KUKA KRL program: MyProgram_106().src

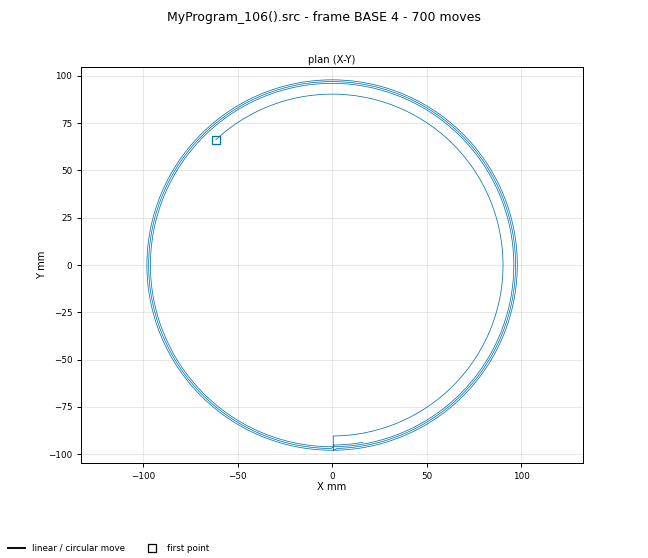
[picture p0: tool path of MyProgram_106().src in frame BASE 4, 700 of 700 moves have a stored position in this frame; points joined in program order, loops and branches not executed]
&ACCESS RVP
&REL 1
&PARAM TEMPLATE = C:\KRC\Roboter\Template\vorgabe
&PARAM EDITMASK = *
DEF MyProgram_106()
; ---- Setting reference (Base) ----
$BASE = BASE_DATA[4]

; --------------------------
; ---- Setting tool (TCP) ----
$TOOL = TOOL_DATA[3]
; --------------------------

$VEL.CP = VEL_APROX_PRINT
Startdeposition()
$VEL.CP = VEL_PRINT
LIN {X -61.5081,Y 66.2185,Z 94,A 127.1384,B 24.9108,C -2.1806,E1 24.8923,E2 -42.0687} C_DIS
LIN {X -59.0339,Y 68.4334,Z 94,A 125.0218,B 24.9104,C -2.1851,E1 24.8968,E2 -39.9543} C_DIS
LIN {X -56.4801,Y 70.5559,Z 94,A 122.9034,B 24.9101,C -2.1892,E1 24.9013,E2 -37.8379} C_DIS
LIN {X -54.0546,Y 72.4294,Z 94,A 121.1393,B 24.9093,C -2.1987,E1 24.9052,E2 -36.09} C_DIS
LIN {X -51.3564,Y 74.3668,Z 94,A 119.0568,B 24.9089,C -2.2037,E1 24.91,E2 -34.012} C_DIS
LIN {X -49.519,Y 75.6028,Z 94,A 117.6469,B 24.9087,C -2.2062,E1 24.9132,E2 -32.6035} C_DIS
LIN {X -47.5461,Y 76.8594,Z 94,A 115.9946,B 24.9089,C -2.2038,E1 24.9172,E2 -30.9403} C_DIS
LIN {X -44.7585,Y 78.515,Z 94,A 113.9269,B 24.9086,C -2.2071,E1 24.9222,E2 -28.8743} C_DIS
LIN {X -41.8485,Y 80.1038,Z 94,A 111.9477,B 24.908,C -2.2144,E1 24.927,E2 -26.9069} C_DIS
LIN {X -39.6316,Y 81.2248,Z 94,A 110.4097,B 24.9077,C -2.218,E1 24.9308,E2 -25.3735} C_DIS
LIN {X -36.8751,Y 82.5114,Z 94,A 108.4363,B 24.9076,C -2.2196,E1 24.9358,E2 -23.3989} C_DIS
LIN {X -34.5929,Y 83.4953,Z 94,A 106.888,B 24.9073,C -2.2227,E1 24.9398,E2 -21.8544} C_DIS
LIN {X -32.7956,Y 84.2161,Z 94,A 105.623,B 24.9073,C -2.2232,E1 24.9431,E2 -20.5879} C_DIS
LIN {X -29.6593,Y 85.3712,Z 94,A 103.3582,B 24.9074,C -2.2214,E1 24.9491,E2 -18.3142} C_DIS
LIN {X -26.4788,Y 86.4106,Z 94,A 101.4259,B 24.9067,C -2.2297,E1 24.9542,E2 -16.3983} C_DIS
LIN {X -24.0911,Y 87.1077,Z 94,A 99.8258,B 24.9067,C -2.2306,E1 24.9585,E2 -14.7978} C_DIS
LIN {X -21.1443,Y 87.8683,Z 94,A 97.8908,B 24.9065,C -2.2324,E1 24.9637,E2 -12.8641} C_DIS
LIN {X -18.7193,Y 88.4179,Z 94,A 96.311,B 24.9065,C -2.2336,E1 24.968,E2 -11.2853} C_DIS
LIN {X -16.8191,Y 88.7977,Z 94,A 95.0427,B 24.9065,C -2.2334,E1 24.9715,E2 -10.015} C_DIS
LIN {X -14.6242,Y 89.1855,Z 94,A 93.4958,B 24.9067,C -2.2302,E1 24.9758,E2 -8.4591} C_DIS
LIN {X -11.3226,Y 89.6645,Z 94,A 91.5124,B 24.9062,C -2.2356,E1 24.9812,E2 -6.4871} C_DIS
LIN {X -8.8533,Y 89.9431,Z 94,A 89.9727,B 24.9061,C -2.2376,E1 24.9855,E2 -4.9513} C_DIS
LIN {X -6.6558,Y 90.1323,Z 94,A 88.571,B 24.9061,C -2.2381,E1 24.9894,E2 -3.5501} C_DIS
LIN {X -4.1214,Y 90.2824,Z 94,A 86.8039,B 24.9064,C -2.2337,E1 24.9944,E2 -1.772} C_DIS
LIN {X -1.0898,Y 90.3711,Z 94,A 84.8009,B 24.9066,C -2.2316,E1 25,E2 0.2361} C_DIS
LIN {X 2.2165,Y 90.3505,Z 94,A 82.9393,B 24.9059,C -2.2394,E1 25.0051,E2 2.0789} C_DIS
LIN {X 5.279,Y 90.2222,Z 94,A 80.9608,B 24.906,C -2.2384,E1 25.0106,E2 4.0591} C_DIS
LIN {X 8.157,Y 90.0073,Z 94,A 79.047,B 24.9062,C -2.2356,E1 25.016,E2 5.9787} C_DIS
LIN {X 10.7987,Y 89.7291,Z 94,A 77.4482,B 24.906,C -2.2381,E1 25.0204,E2 7.5704} C_DIS
LIN {X 12.992,Y 89.4378,Z 94,A 75.9187,B 24.9064,C -2.2336,E1 25.0246,E2 9.1093} C_DIS
LIN {X 16.1999,Y 88.9125,Z 94,A 73.9645,B 24.9062,C -2.2363,E1 25.03,E2 11.0548} C_DIS
LIN {X 19.5413,Y 88.2386,Z 94,A 71.8741,B 24.9061,C -2.2377,E1 25.0357,E2 13.1395} C_DIS
LIN {X 21.9634,Y 87.6684,Z 94,A 70.2868,B 24.9061,C -2.2364,E1 25.04,E2 14.7274} C_DIS
LIN {X 24.9051,Y 86.8772,Z 94,A 68.3251,B 24.9064,C -2.2342,E1 25.0453,E2 16.6913} C_DIS
LIN {X 27.5626,Y 86.071,Z 94,A 66.4674,B 24.9067,C -2.2296,E1 25.0503,E2 18.5565} C_DIS
LIN {X 30.7614,Y 84.9801,Z 94,A 64.315,B 24.9069,C -2.2274,E1 25.0559,E2 20.7098} C_DIS
LIN {X 33.4831,Y 83.946,Z 94,A 62.6281,B 24.9066,C -2.2309,E1 25.0603,E2 22.3847} C_DIS
LIN {X 35.6162,Y 83.0639,Z 94,A 60.9576,B 24.9074,C -2.2224,E1 25.0646,E2 24.0714} C_DIS
LIN {X 38.6404,Y 81.701,Z 94,A 59.0613,B 24.907,C -2.2269,E1 25.0694,E2 25.9522} C_DIS
LIN {X 41.3681,Y 80.3529,Z 94,A 57.1008,B 24.9073,C -2.2234,E1 25.0743,E2 27.9156} C_DIS
LIN {X 43.3395,Y 79.307,Z 94,A 55.5648,B 24.9078,C -2.2174,E1 25.0781,E2 29.4615} C_DIS
LIN {X 46.2751,Y 77.6309,Z 94,A 53.5477,B 24.9077,C -2.2186,E1 25.083,E2 31.4697} C_DIS
LIN {X 48.3763,Y 76.3403,Z 94,A 52.0379,B 24.9077,C -2.218,E1 25.0865,E2 32.9761} C_DIS
LIN {X 50.2205,Y 75.1401,Z 94,A 50.6472,B 24.9079,C -2.2159,E1 25.0898,E2 34.367} C_DIS
LIN {X 52.2581,Y 73.7361,Z 94,A 48.9167,B 24.9086,C -2.2078,E1 25.0938,E2 36.1109} C_DIS
LIN {X 54.6991,Y 71.9452,Z 94,A 46.9487,B 24.909,C -2.2027,E1 25.0982,E2 38.0837} C_DIS
LIN {X 57.3349,Y 69.8631,Z 94,A 44.8265,B 24.9093,C -2.199,E1 25.1028,E2 40.2067} C_DIS
LIN {X 59.8757,Y 67.698,Z 94,A 42.7258,B 24.9096,C -2.1954,E1 25.1072,E2 42.3076} C_DIS
LIN {X 62.3215,Y 65.4535,Z 94,A 40.629,B 24.9099,C -2.1914,E1 25.1115,E2 44.4054} C_DIS
LIN {X 64.6833,Y 63.1206,Z 94,A 38.534,B 24.9103,C -2.1872,E1 25.1156,E2 46.5013} C_DIS
LIN {X 66.9576,Y 60.7026,Z 94,A 36.4373,B 24.9106,C -2.1828,E1 25.1196,E2 48.5992} C_DIS
LIN {X 69.1579,Y 58.1834,Z 94,A 34.3106,B 24.911,C -2.1777,E1 25.1235,E2 50.7283} C_DIS
LIN {X 71.2845,Y 55.5572,Z 94,A 32.1828,B 24.9114,C -2.1731,E1 25.1271,E2 52.8571} C_DIS
LIN {X 73.4267,Y 52.6916,Z 94,A 30.0253,B 24.9116,C -2.1714,E1 25.1307,E2 55.0081} C_DIS
LIN {X 74.9959,Y 50.4334,Z 94,A 28.4236,B 24.9116,C -2.172,E1 25.1332,E2 56.6006} C_DIS
LIN {X 76.2091,Y 48.5808,Z 94,A 27.0277,B 24.9118,C -2.1687,E1 25.1353,E2 57.9974} C_DIS
LIN {X 77.3765,Y 46.6989,Z 94,A 25.6013,B 24.9122,C -2.1642,E1 25.1374,E2 59.4271} C_DIS
LIN {X 78.5152,Y 44.7582,Z 94,A 24.0499,B 24.9128,C -2.1559,E1 25.1396,E2 60.99} C_DIS
LIN {X 80.1014,Y 41.8532,Z 94,A 22.1266,B 24.9128,C -2.1564,E1 25.1421,E2 62.902} C_DIS
LIN {X 81.2217,Y 39.638,Z 94,A 20.3536,B 24.9137,C -2.1449,E1 25.1443,E2 64.6927} C_DIS
LIN {X 82.5072,Y 36.8844,Z 94,A 18.4926,B 24.914,C -2.1418,E1 25.1465,E2 66.5508} C_DIS
LIN {X 83.7784,Y 33.8975,Z 94,A 16.5874,B 24.914,C -2.1413,E1 25.1485,E2 68.4467} C_DIS
LIN {X 84.7137,Y 31.4916,Z 94,A 14.978,B 24.9143,C -2.1375,E1 25.1501,E2 70.0562} C_DIS
LIN {X 85.8199,Y 28.3386,Z 94,A 12.8796,B 24.9148,C -2.1319,E1 25.152,E2 72.1559} C_DIS
LIN {X 86.7244,Y 25.4319,Z 94,A 10.924,B 24.9153,C -2.1252,E1 25.1536,E2 74.1162} C_DIS
LIN {X 87.3926,Y 23.0362,Z 94,A 9.2221,B 24.916,C -2.1159,E1 25.1549,E2 75.8303} C_DIS
LIN {X 88.1253,Y 20.0464,Z 94,A 7.4136,B 24.9161,C -2.1151,E1 25.156,E2 77.6303} C_DIS
LIN {X 88.6437,Y 17.6188,Z 94,A 5.8952,B 24.9163,C -2.1122,E1 25.1569,E2 79.1467} C_DIS
LIN {X 89.0428,Y 15.4757,Z 94,A 4.5192,B 24.9167,C -2.1081,E1 25.1576,E2 80.5244} C_DIS
LIN {X 89.399,Y 13.2645,Z 94,A 3.1049,B 24.917,C -2.1038,E1 25.1582,E2 81.9404} C_DIS
LIN {X 89.6657,Y 11.3128,Z 94,A 1.8305,B 24.9174,C -2.099,E1 25.1587,E2 83.2187} C_DIS
LIN {X 89.943,Y 8.8544,Z 94,A 0.2027,B 24.9179,C -2.0918,E1 25.1591,E2 84.8538} C_DIS
LIN {X 90.197,Y 5.7001,Z 94,A -1.8462,B 24.9186,C -2.0839,E1 25.1595,E2 86.9092} C_DIS
LIN {X 90.3415,Y 2.5118,Z 94,A -3.7689,B 24.9188,C -2.0811,E1 25.1597,E2 88.8271} C_DIS
LIN {X 90.3738,Y -0.7138,Z 94,A -5.9406,B 24.9196,C -2.07,E1 25.1597,E2 91.0121} C_DIS
LIN {X 90.2796,Y -4.186,Z 94,A -7.911,B 24.9196,C -2.0712,E1 25.1596,E2 92.9678} C_DIS
LIN {X 90.1322,Y -6.657,Z 94,A -9.4653,B 24.9199,C -2.0667,E1 25.1593,E2 94.5235} C_DIS
LIN {X 89.9431,Y -8.8525,Z 94,A -10.8563,B 24.9202,C -2.0624,E1 25.1589,E2 95.9164} C_DIS
LIN {X 89.5538,Y -12.1755,Z 94,A -12.9566,B 24.9207,C -2.0564,E1 25.1582,E2 98.0186} C_DIS
LIN {X 89.0487,Y -15.4423,Z 94,A -15.0435,B 24.9212,C -2.05,E1 25.1573,E2 100.1083} C_DIS
LIN {X 88.6386,Y -17.6444,Z 94,A -16.6575,B 24.9221,C -2.0385,E1 25.1564,E2 101.7401} C_DIS
LIN {X 87.933,Y -20.8787,Z 94,A -18.6638,B 24.9223,C -2.0351,E1 25.1552,E2 103.7426} C_DIS
LIN {X 87.1809,Y -23.82,Z 94,A -20.455,B 24.9224,C -2.0339,E1 25.1539,E2 105.5265} C_DIS
LIN {X 86.4846,Y -26.2404,Z 94,A -22.0353,B 24.9228,C -2.0294,E1 25.1527,E2 107.1083} C_DIS
LIN {X 85.8159,Y -28.3509,Z 94,A -23.4299,B 24.9231,C -2.0254,E1 25.1515,E2 108.5045} C_DIS
LIN {X 85.0617,Y -30.5377,Z 94,A -24.8793,B 24.9234,C -2.0214,E1 25.1501,E2 109.955} C_DIS
LIN {X 84.199,Y -32.8392,Z 94,A -26.5824,B 24.9241,C -2.0114,E1 25.1484,E2 111.6723} C_DIS
LIN {X 83.1636,Y -35.3801,Z 94,A -28.1431,B 24.9241,C -2.0126,E1 25.1467,E2 113.2217} C_DIS
LIN {X 82.1671,Y -37.6391,Z 94,A -29.8413,B 24.9248,C -2.003,E1 25.1448,E2 114.9332} C_DIS
LIN {X 80.8611,Y -40.3655,Z 94,A -31.6269,B 24.9248,C -2.002,E1 25.1426,E2 116.7115} C_DIS
LIN {X 79.7039,Y -42.6077,Z 94,A -33.2085,B 24.9252,C -1.998,E1 25.1406,E2 118.2944} C_DIS
LIN {X 78.6361,Y -44.5478,Z 94,A -34.6056,B 24.9254,C -1.9941,E1 25.1387,E2 119.6933} C_DIS
LIN {X 77.6608,Y -46.2246,Z 94,A -35.871,B 24.9258,C -1.9893,E1 25.1369,E2 120.9635} C_DIS
LIN {X 76.3474,Y -48.3653,Z 94,A -37.6069,B 24.9265,C -1.9796,E1 25.1343,E2 122.7135} C_DIS
LIN {X 74.5206,Y -51.1353,Z 94,A -39.4997,B 24.9264,C -1.9813,E1 25.1313,E2 124.593} C_DIS
LIN {X 73.2465,Y -52.9442,Z 94,A -40.8949,B 24.9267,C -1.9777,E1 25.1291,E2 125.9899} C_DIS
LIN {X 71.5903,Y -55.1603,Z 94,A -42.7617,B 24.9273,C -1.969,E1 25.1259,E2 127.8684} C_DIS
LIN {X 69.4989,Y -57.7731,Z 94,A -44.8582,B 24.9277,C -1.9643,E1 25.1222,E2 129.9663} C_DIS
LIN {X 67.3324,Y -60.2842,Z 94,A -46.927,B 24.928,C -1.9601,E1 25.1184,E2 132.0357} C_DIS
LIN {X 65.0939,Y -62.6947,Z 94,A -49.0471,B 24.9284,C -1.9537,E1 25.1143,E2 134.1617} C_DIS
LIN {X 62.7061,Y -65.0829,Z 94,A -51.1535,B 24.9287,C -1.9497,E1 25.1101,E2 136.2685} C_DIS
LIN {X 60.2762,Y -67.3396,Z 94,A -53.2426,B 24.9291,C -1.9453,E1 25.1058,E2 138.3597} C_DIS
LIN {X 57.7644,Y -69.5061,Z 94,A -55.3481,B 24.9294,C -1.9405,E1 25.1013,E2 140.4684} C_DIS
LIN {X 55.1537,Y -71.5954,Z 94,A -57.4017,B 24.9296,C -1.9382,E1 25.0968,E2 142.5197} C_DIS
LIN {X 52.9367,Y -73.2519,Z 94,A -59.0802,B 24.9296,C -1.9372,E1 25.0931,E2 144.1946} C_DIS
LIN {X 50.4391,Y -74.9921,Z 94,A -61.0056,B 24.9299,C -1.9335,E1 25.0886,E2 146.1223} C_DIS
LIN {X 48.5883,Y -76.2043,Z 94,A -62.4025,B 24.9301,C -1.931,E1 25.0854,E2 147.5205} C_DIS
LIN {X 46.7085,Y -77.3707,Z 94,A -63.8378,B 24.9304,C -1.9272,E1 25.0819,E2 148.9603} C_DIS
LIN {X 44.7808,Y -78.5022,Z 94,A -65.3722,B 24.9308,C -1.9206,E1 25.0782,E2 150.5057} C_DIS
LIN {X 41.7682,Y -80.1461,Z 94,A -67.5477,B 24.9311,C -1.9168,E1 25.0728,E2 152.6839} C_DIS
LIN {X 38.8458,Y -81.6023,Z 94,A -69.4397,B 24.9309,C -1.9197,E1 25.0681,E2 154.5642} C_DIS
LIN {X 36.8543,Y -82.5208,Z 94,A -70.8602,B 24.9311,C -1.9165,E1 25.0645,E2 155.9887} C_DIS
LIN {X 34.7762,Y -83.418,Z 94,A -72.2755,B 24.9312,C -1.915,E1 25.0609,E2 157.404} C_DIS
LIN {X 32.799,Y -84.2148,Z 94,A -73.6475,B 24.9314,C -1.9125,E1 25.0573,E2 158.779} C_DIS
LIN {X 29.6525,Y -85.3736,Z 94,A -75.7581,B 24.9316,C -1.9102,E1 25.0517,E2 160.8906} C_DIS
LIN {X 26.4961,Y -86.4053,Z 94,A -77.8241,B 24.9316,C -1.909,E1 25.0462,E2 162.9556} C_DIS
LIN {X 23.8023,Y -87.1857,Z 94,A -79.7527,B 24.9322,C -1.9019,E1 25.041,E2 164.8977} C_DIS
LIN {X 21.128,Y -87.8722,Z 94,A -81.344,B 24.9319,C -1.9056,E1 25.0367,E2 166.478} C_DIS
LIN {X 18.7084,Y -88.4202,Z 94,A -82.9114,B 24.932,C -1.9043,E1 25.0325,E2 168.0464} C_DIS
LIN {X 16.8115,Y -88.7991,Z 94,A -84.1698,B 24.9322,C -1.9022,E1 25.029,E2 169.3083} C_DIS
LIN {X 14.637,Y -89.1833,Z 94,A -85.5783,B 24.9322,C -1.9009,E1 25.0251,E2 170.7185} C_DIS
LIN {X 12.1543,Y -89.5567,Z 94,A -87.1203,B 24.9322,C -1.9014,E1 25.0209,E2 172.2578} C_DIS
LIN {X 9.66,Y -89.8587,Z 94,A -88.873,B 24.9327,C -1.8951,E1 25.016,E2 174.0241} C_DIS
LIN {X 6.7485,Y -90.1249,Z 94,A -90.5759,B 24.9324,C -1.8992,E1 25.0113,E2 175.7165} C_DIS
LIN {X 3.9373,Y -90.2903,Z 94,A -92.4515,B 24.9326,C -1.8955,E1 25.006,E2 177.6002} C_DIS
LIN {X 0.6412,Y -90.373,Z 94,A -94.5139,B 24.9326,C -1.8959,E1 25.0003,E2 179.6615} C_DIS
Enddeposition()
LIN {X 0.6684,Y -97.9224,Z 95,A -93.7838,B 24.9395,C -1.7963,E1 25.0016,E2 179.1676} C_DIS
Startdeposition()
$VEL.CP = VEL_PRINT
LIN {X -2.4033,Y -97.8979,Z 95,A -95.9763,B 24.9405,C -1.7815,E1 24.9954,E2 181.3953} C_DIS
LIN {X -4.6034,Y -97.8181,Z 95,A -97.2798,B 24.9405,C -1.7808,E1 24.9918,E2 182.7006} C_DIS
LIN {X -7.0026,Y -97.6757,Z 95,A -98.686,B 24.9405,C -1.7808,E1 24.9878,E2 184.1074} C_DIS
LIN {X -9.3975,Y -97.4744,Z 95,A -100.0925,B 24.9405,C -1.7808,E1 24.9839,E2 185.5144} C_DIS
LIN {X -11.7401,Y -97.2199,Z 95,A -101.461,B 24.9405,C -1.7814,E1 24.9801,E2 186.8825} C_DIS
LIN {X -14.1691,Y -96.8959,Z 95,A -102.9063,B 24.9405,C -1.7813,E1 24.9761,E2 188.3292} C_DIS
LIN {X -16.5427,Y -96.519,Z 95,A -104.2975,B 24.9405,C -1.7822,E1 24.9723,E2 189.7195} C_DIS
LIN {X -18.9064,Y -96.084,Z 95,A -105.7048,B 24.9405,C -1.7827,E1 24.9684,E2 191.1271} C_DIS
LIN {X -21.456,Y -95.548,Z 95,A -107.4483,B 24.9409,C -1.7756,E1 24.9636,E2 192.8896} C_DIS
LIN {X -24.9583,Y -94.6935,Z 95,A -109.5462,B 24.9409,C -1.7772,E1 24.958,E2 194.9868} C_DIS
LIN {X -28.2333,Y -93.7681,Z 95,A -111.3527,B 24.9403,C -1.7851,E1 24.9532,E2 196.7775} C_DIS
LIN {X -30.718,Y -92.9849,Z 95,A -112.8638,B 24.9402,C -1.7867,E1 24.9491,E2 198.2875} C_DIS
LIN {X -32.8003,Y -92.2698,Z 95,A -114.1543,B 24.9401,C -1.7878,E1 24.9457,E2 199.578} C_DIS
LIN {X -35.0548,Y -91.4371,Z 95,A -115.5725,B 24.9401,C -1.7886,E1 24.942,E2 200.9972} C_DIS
LIN {X -37.6613,Y -90.3948,Z 95,A -117.3562,B 24.9403,C -1.7853,E1 24.9374,E2 202.7926} C_DIS
LIN {X -40.7799,Y -89.0325,Z 95,A -119.2055,B 24.9398,C -1.7924,E1 24.9327,E2 204.6295} C_DIS
LIN {X -43.6727,Y -87.6479,Z 95,A -121.1405,B 24.9398,C -1.7927,E1 24.9278,E2 206.5689} C_DIS
LIN {X -45.984,Y -86.4584,Z 95,A -122.6279,B 24.9396,C -1.7958,E1 24.9242,E2 208.053} C_DIS
LIN {X -48.2683,Y -85.2054,Z 95,A -124.1407,B 24.9394,C -1.7983,E1 24.9205,E2 209.5644} C_DIS
LIN {X -50.171,Y -84.0979,Z 95,A -125.4331,B 24.9393,C -1.8,E1 24.9174,E2 210.8566} C_DIS
LIN {X -52.2197,Y -82.8413,Z 95,A -126.8458,B 24.9391,C -1.8019,E1 24.914,E2 212.2692} C_DIS
LIN {X -54.4056,Y -81.4237,Z 95,A -128.3735,B 24.939,C -1.8041,E1 24.9105,E2 213.7965} C_DIS
LIN {X -56.2216,Y -80.1792,Z 95,A -129.6664,B 24.9389,C -1.8061,E1 24.9075,E2 215.0892} C_DIS
LIN {X -58.3353,Y -78.6561,Z 95,A -131.1964,B 24.9387,C -1.8085,E1 24.904,E2 216.6188} C_DIS
LIN {X -60.2481,Y -77.2007,Z 95,A -132.8207,B 24.939,C -1.8036,E1 24.9004,E2 218.2607} C_DIS
LIN {X -62.8149,Y -75.1252,Z 95,A -134.5809,B 24.9384,C -1.813,E1 24.8966,E2 220.0052} C_DIS
LIN {X -64.8687,Y -73.361,Z 95,A -136.1387,B 24.9381,C -1.817,E1 24.8934,E2 221.5597} C_DIS
LIN {X -66.5008,Y -71.8835,Z 95,A -137.4483,B 24.938,C -1.8188,E1 24.8907,E2 222.8701} C_DIS
LIN {X -68.2448,Y -70.2298,Z 95,A -138.8401,B 24.9378,C -1.8222,E1 24.8879,E2 224.2597} C_DIS
LIN {X -69.9478,Y -68.5338,Z 95,A -140.2449,B 24.9376,C -1.8253,E1 24.8851,E2 225.6632} C_DIS
LIN {X -71.6086,Y -66.7966,Z 95,A -141.6446,B 24.9373,C -1.8285,E1 24.8824,E2 227.0612} C_DIS
LIN {X -73.2263,Y -65.0191,Z 95,A -143.0841,B 24.9372,C -1.8306,E1 24.8797,E2 228.5023} C_DIS
LIN {X -74.7999,Y -63.2025,Z 95,A -144.513,B 24.937,C -1.833,E1 24.8771,E2 229.9317} C_DIS
LIN {X -76.4556,Y -61.1909,Z 95,A -146.0294,B 24.9368,C -1.8369,E1 24.8745,E2 231.4461} C_DIS
LIN {X -77.9343,Y -59.2961,Z 95,A -147.4434,B 24.9365,C -1.84,E1 24.8721,E2 232.8594} C_DIS
LIN {X -79.2467,Y -57.5286,Z 95,A -148.754,B 24.9364,C -1.8424,E1 24.8699,E2 234.1705} C_DIS
LIN {X -80.7499,Y -55.4007,Z 95,A -150.2713,B 24.9361,C -1.8465,E1 24.8675,E2 235.6856} C_DIS
LIN {X -81.9741,Y -53.5708,Z 95,A -151.5663,B 24.9359,C -1.8495,E1 24.8655,E2 236.9798} C_DIS
LIN {X -83.371,Y -51.3717,Z 95,A -153.3116,B 24.9361,C -1.8462,E1 24.8629,E2 238.742} C_DIS
LIN {X -85.0917,Y -48.4661,Z 95,A -155.0897,B 24.9353,C -1.858,E1 24.8604,E2 240.5012} C_DIS
LIN {X -86.2095,Y -46.448,Z 95,A -156.4824,B 24.9351,C -1.8602,E1 24.8585,E2 241.8959} C_DIS
LIN {X -87.3793,Y -44.2091,Z 95,A -157.9475,B 24.9348,C -1.8647,E1 24.8567,E2 243.3581} C_DIS
LIN {X -88.5254,Y -41.8694,Z 95,A -159.4655,B 24.9345,C -1.8692,E1 24.8548,E2 244.8736} C_DIS
LIN {X -89.4433,Y -39.8683,Z 95,A -160.7617,B 24.9343,C -1.8726,E1 24.8533,E2 246.1688} C_DIS
LIN {X -90.3948,Y -37.6613,Z 95,A -162.1929,B 24.934,C -1.8758,E1 24.8518,E2 247.6003} C_DIS
LIN {X -91.2918,Y -35.4315,Z 95,A -163.608,B 24.9338,C -1.8796,E1 24.8503,E2 249.0143} C_DIS
LIN {X -92.1646,Y -33.0961,Z 95,A -165.0655,B 24.9335,C -1.8839,E1 24.8489,E2 250.4698} C_DIS
LIN {X -92.9204,Y -30.9094,Z 95,A -166.4229,B 24.9332,C -1.8878,E1 24.8477,E2 251.8255} C_DIS
LIN {X -93.6509,Y -28.6197,Z 95,A -167.8425,B 24.9329,C -1.8916,E1 24.8465,E2 253.2443} C_DIS
LIN {X -94.3801,Y -26.1185,Z 95,A -169.3729,B 24.9326,C -1.896,E1 24.8454,E2 254.773} C_DIS
LIN {X -94.9063,Y -24.1304,Z 95,A -170.6045,B 24.9324,C -1.8988,E1 24.8445,E2 256.0052} C_DIS
LIN {X -95.548,Y -21.456,Z 95,A -172.2043,B 24.932,C -1.904,E1 24.8435,E2 257.602} C_DIS
LIN {X -96.0458,Y -19.1047,Z 95,A -173.6204,B 24.9317,C -1.9081,E1 24.8427,E2 259.0168} C_DIS
LIN {X -96.6839,Y -15.5566,Z 95,A -175.7437,B 24.9313,C -1.9142,E1 24.8417,E2 261.138} C_DIS
LIN {X -97.0366,Y -13.1791,Z 95,A -177.16,B 24.931,C -1.9183,E1 24.8411,E2 262.5529} C_DIS
LIN {X -97.3308,Y -10.7938,Z 95,A -178.5761,B 24.9307,C -1.9224,E1 24.8407,E2 263.9677} C_DIS
LIN {X -97.5663,Y -8.4019,Z 95,A -179.9921,B 24.9304,C -1.9266,E1 24.8403,E2 265.3823} C_DIS
LIN {X -97.7431,Y -6.005,Z 95,A 178.5917,B 24.9301,C -1.9307,E1 24.84,E2 266.7971} C_DIS
LIN {X -97.8611,Y -3.6044,Z 95,A 177.1757,B 24.9298,C -1.9349,E1 24.8399,E2 268.2116} C_DIS
LIN {X -97.922,Y -0.9299,Z 95,A 175.4202,B 24.9298,C -1.9338,E1 24.8398,E2 269.9803} C_DIS
LIN {X -97.8979,Y 2.4033,Z 95,A 173.6349,B 24.929,C -1.9454,E1 24.8398,E2 271.7488} C_DIS
LIN {X -97.8181,Y 4.6034,Z 95,A 172.3233,B 24.9288,C -1.9488,E1 24.84,E2 273.0602} C_DIS
LIN {X -97.6757,Y 7.0026,Z 95,A 170.9056,B 24.9285,C -1.9529,E1 24.8403,E2 274.4765} C_DIS
LIN {X -97.4744,Y 9.3975,Z 95,A 169.4894,B 24.9282,C -1.9571,E1 24.8406,E2 275.8912} C_DIS
LIN {X -97.2145,Y 11.7868,Z 95,A 168.089,B 24.9278,C -1.9618,E1 24.8411,E2 277.2888} C_DIS
LIN {X -96.8959,Y 14.1691,Z 95,A 166.6571,B 24.9276,C -1.9655,E1 24.8416,E2 278.7205} C_DIS
LIN {X -96.519,Y 16.5427,Z 95,A 165.2566,B 24.9272,C -1.9702,E1 24.8423,E2 280.118} C_DIS
LIN {X -96.1378,Y 18.6269,Z 95,A 163.9576,B 24.9271,C -1.9722,E1 24.8429,E2 281.4198} C_DIS
LIN {X -95.548,Y 21.456,Z 95,A 162.3056,B 24.9266,C -1.9788,E1 24.8439,E2 283.0658} C_DIS
LIN {X -94.7438,Y 24.7628,Z 95,A 160.2846,B 24.9262,C -1.9842,E1 24.8453,E2 285.0859} C_DIS
LIN {X -94.1075,Y 27.0805,Z 95,A 158.8845,B 24.9258,C -1.9888,E1 24.8463,E2 286.483} C_DIS
LIN {X -93.3548,Y 29.5747,Z 95,A 157.3497,B 24.9255,C -1.9932,E1 24.8476,E2 288.0162} C_DIS
LIN {X -92.203,Y 32.9908,Z 95,A 155.2258,B 24.9251,C -1.9993,E1 24.8495,E2 290.1377} C_DIS
LIN {X -90.9262,Y 36.3621,Z 95,A 153.1024,B 24.9246,C -2.0053,E1 24.8516,E2 292.2587} C_DIS
LIN {X -90.0849,Y 38.3966,Z 95,A 151.8055,B 24.9243,C -2.009,E1 24.853,E2 293.5541} C_DIS
LIN {X -89.2516,Y 40.2937,Z 95,A 150.4959,B 24.9243,C -2.0095,E1 24.8545,E2 294.8697} C_DIS
LIN {X -88.0923,Y 42.7706,Z 95,A 148.9584,B 24.9238,C -2.0163,E1 24.8564,E2 296.3993} C_DIS
LIN {X -87.0162,Y 44.9196,Z 95,A 147.5431,B 24.9235,C -2.0201,E1 24.8582,E2 297.813} C_DIS
LIN {X -85.7913,Y 47.219,Z 95,A 145.8069,B 24.9237,C -2.0177,E1 24.8605,E2 299.5642} C_DIS
LIN {X -84.0979,Y 50.171,Z 95,A 144.0052,B 24.9228,C -2.0296,E1 24.863,E2 301.3469} C_DIS
LIN {X -82.7343,Y 52.3909,Z 95,A 142.4869,B 24.9224,C -2.0341,E1 24.8652,E2 302.8622} C_DIS
LIN {X -81.5348,Y 54.237,Z 95,A 141.1751,B 24.9222,C -2.0369,E1 24.8673,E2 304.1738} C_DIS
LIN {X -80.1792,Y 56.2216,Z 95,A 139.7897,B 24.9219,C -2.0414,E1 24.8695,E2 305.5552} C_DIS
LIN {X -78.6561,Y 58.3353,Z 95,A 138.2428,B 24.9216,C -2.0448,E1 24.872,E2 307.1016} C_DIS
LIN {X -77.324,Y 60.0881,Z 95,A 136.9312,B 24.9214,C -2.0475,E1 24.8742,E2 308.4131} C_DIS
LIN {X -75.8261,Y 61.9677,Z 95,A 135.517,B 24.9211,C -2.0509,E1 24.8767,E2 309.8257} C_DIS
LIN {X -74.1553,Y 63.9591,Z 95,A 134.0031,B 24.9208,C -2.0551,E1 24.8794,E2 311.3366} C_DIS
LIN {X -72.6984,Y 65.6088,Z 95,A 132.6916,B 24.9206,C -2.0575,E1 24.8819,E2 312.648} C_DIS
LIN {X -70.9237,Y 67.5249,Z 95,A 131.1715,B 24.9203,C -2.0616,E1 24.8848,E2 314.1652} C_DIS
LIN {X -69.387,Y 69.1015,Z 95,A 129.8766,B 24.9201,C -2.0645,E1 24.8873,E2 315.4586} C_DIS
LIN {X -67.5249,Y 70.9237,Z 95,A 128.3446,B 24.9198,C -2.0678,E1 24.8904,E2 316.9891} C_DIS
LIN {X -65.0191,Y 73.2263,Z 95,A 126.3271,B 24.9195,C -2.0716,E1 24.8946,E2 319.0058} C_DIS
LIN {X -63.0488,Y 74.9309,Z 95,A 124.8113,B 24.9192,C -2.0752,E1 24.8978,E2 320.5187} C_DIS
LIN {X -61.1909,Y 76.4556,Z 95,A 123.3981,B 24.919,C -2.0781,E1 24.9008,E2 321.9305} C_DIS
LIN {X -59.4561,Y 77.811,Z 95,A 122.0882,B 24.9189,C -2.0801,E1 24.9037,E2 323.2404} C_DIS
LIN {X -56.3874,Y 80.064,Z 95,A 119.8664,B 24.9185,C -2.0848,E1 24.9087,E2 325.4587} C_DIS
LIN {X -54.5727,Y 81.3105,Z 95,A 118.5572,B 24.9183,C -2.0866,E1 24.9118,E2 326.7679} C_DIS
LIN {X -51.872,Y 83.0585,Z 95,A 116.6046,B 24.9183,C -2.0879,E1 24.9164,E2 328.7239} C_DIS
LIN {X -49.484,Y 84.5039,Z 95,A 115.0269,B 24.9179,C -2.0927,E1 24.9201,E2 330.295} C_DIS
LIN {X -46.3401,Y 86.268,Z 95,A 112.9097,B 24.9176,C -2.096,E1 24.9253,E2 332.4102} C_DIS
LIN {X -44.2091,Y 87.3793,Z 95,A 111.5143,B 24.9174,C -2.0987,E1 24.9288,E2 333.803} C_DIS
LIN {X -41.8694,Y 88.5254,Z 95,A 109.9847,B 24.9172,C -2.1009,E1 24.9326,E2 335.3313} C_DIS
LIN {X -38.97,Y 89.8376,Z 95,A 108.0807,B 24.9172,C -2.1023,E1 24.9375,E2 337.2367} C_DIS
LIN {X -36.5491,Y 90.8501,Z 95,A 106.5764,B 24.9169,C -2.1055,E1 24.9413,E2 338.7367} C_DIS
LIN {X -34.1197,Y 91.7912,Z 95,A 105.0475,B 24.9167,C -2.1073,E1 24.9453,E2 340.2644} C_DIS
LIN {X -31.8568,Y 92.6009,Z 95,A 103.6375,B 24.9166,C -2.1089,E1 24.949,E2 341.6733} C_DIS
LIN {X -28.6197,Y 93.6509,Z 95,A 101.6253,B 24.9165,C -2.1105,E1 24.9544,E2 343.6854} C_DIS
LIN {X -26.1185,Y 94.3801,Z 95,A 100.1133,B 24.9163,C -2.1126,E1 24.9584,E2 345.195} C_DIS
LIN {X -23.7944,Y 94.9927,Z 95,A 98.7041,B 24.9162,C -2.1139,E1 24.9623,E2 346.6032} C_DIS
LIN {X -21.456,Y 95.548,Z 95,A 97.2948,B 24.9162,C -2.115,E1 24.9661,E2 348.0115} C_DIS
LIN {X -17.9246,Y 96.273,Z 95,A 95.1817,B 24.916,C -2.1166,E1 24.9719,E2 350.1232} C_DIS
LIN {X -15.5566,Y 96.6839,Z 95,A 93.6801,B 24.9162,C -2.1143,E1 24.976,E2 351.6317} C_DIS
LIN {X -12.528,Y 97.1209,Z 95,A 91.8881,B 24.9161,C -2.1154,E1 24.981,E2 353.4224} C_DIS
LIN {X -8.4019,Y 97.5663,Z 95,A 89.5494,B 24.9157,C -2.1198,E1 24.9875,E2 355.7522} C_DIS
LIN {X -6.3464,Y 97.7201,Z 95,A 88.3226,B 24.9157,C -2.1196,E1 24.9909,E2 356.9799} C_DIS
LIN {X -3.6044,Y 97.8611,Z 95,A 86.7347,B 24.9157,C -2.1208,E1 24.9953,E2 358.5653} C_DIS
LIN {X -1.2017,Y 97.9201,Z 95,A 85.3277,B 24.9157,C -2.1211,E1 24.9992,E2 359.9716} C_DIS
LIN {X 1.2017,Y 97.9201,Z 95,A 83.9207,B 24.9157,C -2.1213,E1 25.0032,E2 361.378} C_DIS
LIN {X 3.6044,Y 97.8611,Z 95,A 82.5141,B 24.9156,C -2.1214,E1 25.0071,E2 362.784} C_DIS
LIN {X 6.005,Y 97.7431,Z 95,A 81.1077,B 24.9156,C -2.1214,E1 25.011,E2 364.1898} C_DIS
LIN {X 8.0922,Y 97.5911,Z 95,A 79.8694,B 24.9156,C -2.1209,E1 25.0144,E2 365.4289} C_DIS
LIN {X 10.7938,Y 97.3308,Z 95,A 78.2963,B 24.9156,C -2.1212,E1 25.0188,E2 367.0002} C_DIS
LIN {X 14.3689,Y 96.8675,Z 95,A 76.1875,B 24.9156,C -2.1207,E1 25.0246,E2 369.1083} C_DIS
LIN {X 16.5427,Y 96.519,Z 95,A 74.9003,B 24.9156,C -2.1203,E1 25.0282,E2 370.3952} C_DIS
LIN {X 19.1047,Y 96.0458,Z 95,A 73.3774,B 24.9157,C -2.1198,E1 25.0324,E2 371.9177} C_DIS
LIN {X 21.2588,Y 95.591,Z 95,A 72.0907,B 24.9157,C -2.1192,E1 25.0359,E2 373.2041} C_DIS
LIN {X 23.7902,Y 94.9937,Z 95,A 70.5712,B 24.9158,C -2.1184,E1 25.04,E2 374.7233} C_DIS
LIN {X 26.8552,Y 94.1714,Z 95,A 68.6783,B 24.916,C -2.1159,E1 25.0451,E2 376.619} C_DIS
LIN {X 29.5747,Y 93.3548,Z 95,A 67.0581,B 24.916,C -2.1161,E1 25.0494,E2 378.2358} C_DIS
LIN {X 31.8568,Y 92.6009,Z 95,A 65.6544,B 24.9161,C -2.115,E1 25.0531,E2 379.6394} C_DIS
LIN {X 35.0548,Y 91.4371,Z 95,A 63.6911,B 24.9161,C -2.1142,E1 25.0583,E2 381.6004} C_DIS
LIN {X 37.4752,Y 90.4732,Z 95,A 62.1463,B 24.9164,C -2.1119,E1 25.0623,E2 383.1473} C_DIS
LIN {X 39.4992,Y 89.6069,Z 95,A 60.8462,B 24.9165,C -2.11,E1 25.0656,E2 384.4486} C_DIS
LIN {X 41.6863,Y 88.6106,Z 95,A 59.4586,B 24.9165,C -2.1091,E1 25.0691,E2 385.8349} C_DIS
LIN {X 44.0293,Y 87.4712,Z 95,A 57.9382,B 24.9167,C -2.1073,E1 25.0729,E2 387.3555} C_DIS
LIN {X 45.984,Y 86.4584,Z 95,A 56.6382,B 24.9169,C -2.1052,E1 25.0761,E2 388.6569} C_DIS
LIN {X 48.2683,Y 85.2054,Z 95,A 55.1344,B 24.9169,C -2.1038,E1 25.0798,E2 390.1595} C_DIS
LIN {X 51.3717,Y 83.371,Z 95,A 53.0314,B 24.9172,C -2.1009,E1 25.0848,E2 392.2628} C_DIS
LIN {X 53.4023,Y 82.0852,Z 95,A 51.63,B 24.9174,C -2.0989,E1 25.0881,E2 393.6645} C_DIS
LIN {X 55.2335,Y 80.8631,Z 95,A 50.3466,B 24.9175,C -2.097,E1 25.0911,E2 394.9481} C_DIS
LIN {X 57.2013,Y 79.4833,Z 95,A 48.9297,B 24.9178,C -2.0942,E1 25.0943,E2 396.3666} C_DIS
LIN {X 60.2481,Y 77.2007,Z 95,A 46.7267,B 24.918,C -2.0911,E1 25.0992,E2 398.5689} C_DIS
LIN {X 61.9677,Y 75.8261,Z 95,A 45.4438,B 24.9182,C -2.0889,E1 25.102,E2 399.8521} C_DIS
LIN {X 63.8099,Y 74.2824,Z 95,A 44.0436,B 24.9184,C -2.0864,E1 25.105,E2 401.2527} C_DIS
LIN {X 65.4487,Y 72.8418,Z 95,A 42.7367,B 24.9186,C -2.0828,E1 25.1077,E2 402.5631} C_DIS
LIN {X 67.5249,Y 70.9237,Z 95,A 41.126,B 24.9188,C -2.081,E1 25.111,E2 404.1715} C_DIS
LIN {X 69.1015,Y 69.387,Z 95,A 39.8276,B 24.919,C -2.0779,E1 25.1136,E2 405.4717} C_DIS
LIN {X 70.9237,Y 67.5249,Z 95,A 38.3261,B 24.9192,C -2.0754,E1 25.1165,E2 406.9725} C_DIS
LIN {X 72.5594,Y 65.764,Z 95,A 36.9269,B 24.9194,C -2.0726,E1 25.1192,E2 408.3724} C_DIS
LIN {X 74.0187,Y 64.1156,Z 95,A 35.6452,B 24.9197,C -2.0699,E1 25.1215,E2 409.6547} C_DIS
LIN {X 75.5699,Y 62.2798,Z 95,A 34.2304,B 24.9199,C -2.0663,E1 25.1241,E2 411.0715} C_DIS
LIN {X 77.6027,Y 59.7264,Z 95,A 32.2555,B 24.9205,C -2.0592,E1 25.1275,E2 413.0538} C_DIS
LIN {X 80.064,Y 56.3874,Z 95,A 29.9324,B 24.9206,C -2.0571,E1 25.1313,E2 415.3706} C_DIS
LIN {X 81.4237,Y 54.4056,Z 95,A 28.5339,B 24.9209,C -2.0538,E1 25.1335,E2 416.7699} C_DIS
LIN {X 82.7343,Y 52.3909,Z 95,A 27.1356,B 24.9212,C -2.0505,E1 25.1356,E2 418.1691} C_DIS
LIN {X 83.8903,Y 50.5173,Z 95,A 25.8392,B 24.9214,C -2.0468,E1 25.1375,E2 419.4675} C_DIS
LIN {X 85.2054,Y 48.2683,Z 95,A 24.3393,B 24.9217,C -2.0436,E1 25.1396,E2 420.9673} C_DIS
LIN {X 86.268,Y 46.3401,Z 95,A 23.059,B 24.9219,C -2.0404,E1 25.1413,E2 422.2484} C_DIS
LIN {X 87.4712,Y 44.0293,Z 95,A 21.5437,B 24.9222,C -2.0366,E1 25.1432,E2 423.7648} C_DIS
LIN {X 88.5254,Y 41.8694,Z 95,A 20.1458,B 24.9225,C -2.0329,E1 25.1449,E2 425.1637} C_DIS
LIN {X 90.0065,Y 38.5826,Z 95,A 18.0498,B 24.9229,C -2.0274,E1 25.1473,E2 427.2613} C_DIS
LIN {X 90.9262,Y 36.3621,Z 95,A 16.6521,B 24.9232,C -2.0237,E1 25.1487,E2 428.6601} C_DIS
LIN {X 91.7197,Y 34.3086,Z 95,A 15.3567,B 24.9235,C -2.0196,E1 25.15,E2 429.9578} C_DIS
LIN {X 92.5341,Y 32.0473,Z 95,A 13.9594,B 24.9238,C -2.0158,E1 25.1513,E2 431.3563} C_DIS
LIN {X 93.3548,Y 29.5747,Z 95,A 12.461,B 24.9241,C -2.0122,E1 25.1526,E2 432.8547} C_DIS
LIN {X 93.9491,Y 27.6233,Z 95,A 11.2298,B 24.9245,C -2.0072,E1 25.1536,E2 434.0908} C_DIS
LIN {X 94.6409,Y 25.1532,Z 95,A 9.7841,B 24.9246,C -2.0048,E1 25.1547,E2 435.5339} C_DIS
LIN {X 95.2297,Y 22.8231,Z 95,A 8.3716,B 24.925,C -2.0002,E1 25.1556,E2 436.949} C_DIS
LIN {X 95.7611,Y 20.4791,Z 95,A 6.9748,B 24.9253,C -1.9962,E1 25.1565,E2 438.3471} C_DIS
LIN {X 96.2348,Y 18.1229,Z 95,A 5.5781,B 24.9256,C -1.9922,E1 25.1572,E2 439.7451} C_DIS
LIN {X 96.6506,Y 15.7557,Z 95,A 4.1815,B 24.9259,C -1.9882,E1 25.1579,E2 441.143} C_DIS
LIN {X 97.0366,Y 13.1791,Z 95,A 2.6833,B 24.9262,C -1.9844,E1 25.1585,E2 442.6413} C_DIS
LIN {X 97.3673,Y 10.4444,Z 95,A 0.9643,B 24.9269,C -1.9751,E1 25.159,E2 444.3721} C_DIS
LIN {X 97.646,Y 7.4052,Z 95,A -0.7066,B 24.9269,C -1.9739,E1 25.1594,E2 446.036} C_DIS
LIN {X 97.7983,Y 5.0067,Z 95,A -2.103,B 24.9273,C -1.9698,E1 25.1596,E2 447.4338} C_DIS
LIN {X 97.8918,Y 2.6051,Z 95,A -3.4841,B 24.9275,C -1.9662,E1 25.1597,E2 448.815} C_DIS
LIN {X 97.9263,Y 0.0664,Z 95,A -5.0295,B 24.928,C -1.9591,E1 25.1597,E2 450.368} C_DIS
LIN {X 97.8611,Y -3.6044,Z 95,A -7.0922,B 24.9283,C -1.9555,E1 25.1597,E2 452.4268} C_DIS
LIN {X 97.7431,Y -6.005,Z 95,A -8.4885,B 24.9286,C -1.9514,E1 25.1594,E2 453.8246} C_DIS
LIN {X 97.4744,Y -9.3975,Z 95,A -10.4816,B 24.9291,C -1.9449,E1 25.159,E2 455.8212} C_DIS
LIN {X 97.2145,Y -11.7868,Z 95,A -11.8624,B 24.9293,C -1.9414,E1 25.1585,E2 457.2022} C_DIS
LIN {X 96.9232,Y -13.977,Z 95,A -13.1989,B 24.9298,C -1.9355,E1 25.158,E2 458.5446} C_DIS
LIN {X 96.519,Y -16.5427,Z 95,A -14.6553,B 24.9299,C -1.9331,E1 25.1573,E2 459.9982} C_DIS
LIN {X 96.084,Y -18.9064,Z 95,A -16.1597,B 24.9305,C -1.9247,E1 25.1565,E2 461.5135} C_DIS
LIN {X 95.409,Y -22.058,Z 95,A -18.0268,B 24.9309,C -1.9195,E1 25.1554,E2 463.3822} C_DIS
LIN {X 94.7438,Y -24.7628,Z 95,A -19.5586,B 24.931,C -1.9181,E1 25.1544,E2 464.9083} C_DIS
LIN {X 93.8285,Y -28.0299,Z 95,A -21.5717,B 24.9316,C -1.9108,E1 25.1528,E2 466.9272} C_DIS
LIN {X 92.7998,Y -31.2669,Z 95,A -23.575,B 24.932,C -1.9039,E1 25.1511,E2 468.9353} C_DIS
LIN {X 91.8604,Y -33.9301,Z 95,A -25.1299,B 24.9321,C -1.9026,E1 25.1496,E2 470.4845} C_DIS
LIN {X 90.9262,Y -36.3621,Z 95,A -26.6437,B 24.9324,C -1.8983,E1 25.1481,E2 472.0001} C_DIS
LIN {X 90.0065,Y -38.5826,Z 95,A -28.041,B 24.9327,C -1.8944,E1 25.1465,E2 473.399} C_DIS
LIN {X 89.0325,Y -40.7799,Z 95,A -29.438,B 24.933,C -1.8905,E1 25.1449,E2 474.7977} C_DIS
LIN {X 88.0923,Y -42.7706,Z 95,A -30.7179,B 24.9333,C -1.887,E1 25.1434,E2 476.0789} C_DIS
LIN {X 86.9243,Y -45.0994,Z 95,A -32.2321,B 24.9335,C -1.8828,E1 25.1415,E2 477.5949} C_DIS
LIN {X 85.7913,Y -47.219,Z 95,A -33.6295,B 24.9338,C -1.879,E1 25.1396,E2 478.9939} C_DIS
LIN {X 84.0979,Y -50.171,Z 95,A -35.6082,B 24.9342,C -1.8738,E1 25.1368,E2 480.9748} C_DIS
LIN {X 82.8413,Y -52.2197,Z 95,A -37.0214,B 24.9345,C -1.8695,E1 25.1348,E2 482.391} C_DIS
LIN {X 81.4237,Y -54.4056,Z 95,A -38.5207,B 24.9347,C -1.8662,E1 25.1325,E2 483.8906} C_DIS
LIN {X 79.4833,Y -57.2013,Z 95,A -40.4959,B 24.9351,C -1.8613,E1 25.1293,E2 485.8676} C_DIS
LIN {X 78.0555,Y -59.1347,Z 95,A -41.898,B 24.9353,C -1.8576,E1 25.1269,E2 487.2717} C_DIS
LIN {X 76.5808,Y -61.0325,Z 95,A -43.2963,B 24.9356,C -1.8542,E1 25.1245,E2 488.6715} C_DIS
LIN {X 75.0848,Y -62.8636,Z 95,A -44.6934,B 24.9358,C -1.85,E1 25.122,E2 490.072} C_DIS
LIN {X 73.361,Y -64.8687,Z 95,A -46.2105,B 24.936,C -1.8472,E1 25.1192,E2 491.5889} C_DIS
LIN {X 71.8835,Y -66.5008,Z 95,A -47.5071,B 24.9363,C -1.8436,E1 25.1168,E2 492.8883} C_DIS
LIN {X 70.2298,Y -68.2448,Z 95,A -48.9057,B 24.9365,C -1.8404,E1 25.1141,E2 494.2884} C_DIS
LIN {X 67.5249,Y -70.9237,Z 95,A -51.1057,B 24.9368,C -1.8361,E1 25.1097,E2 496.4895} C_DIS
LIN {X 65.764,Y -72.5594,Z 95,A -52.5047,B 24.937,C -1.8331,E1 25.1068,E2 497.8898} C_DIS
LIN {X 64.1156,Y -74.0187,Z 95,A -53.7866,B 24.9372,C -1.8304,E1 25.1041,E2 499.1731} C_DIS
LIN {X 62.1245,Y -75.6989,Z 95,A -55.3037,B 24.9374,C -1.8272,E1 25.1009,E2 500.6917} C_DIS
LIN {X 60.2481,Y -77.2007,Z 95,A -56.7032,B 24.9376,C -1.8244,E1 25.0978,E2 502.0927} C_DIS
LIN {X 58.3353,Y -78.6561,Z 95,A -58.1027,B 24.9378,C -1.8217,E1 25.0947,E2 503.4936} C_DIS
LIN {X 56.3874,Y -80.064,Z 95,A -59.5029,B 24.938,C -1.8191,E1 25.0915,E2 504.8952} C_DIS
LIN {X 54.4056,Y -81.4237,Z 95,A -60.903,B 24.9382,C -1.8165,E1 25.0882,E2 506.2967} C_DIS
LIN {X 52.5609,Y -82.6253,Z 95,A -62.1582,B 24.9382,C -1.8153,E1 25.0853,E2 507.5506} C_DIS
LIN {X 50.3448,Y -83.9952,Z 95,A -63.7038,B 24.9385,C -1.8116,E1 25.0816,E2 509.1} C_DIS
LIN {X 48.2683,Y -85.2054,Z 95,A -65.1045,B 24.9386,C -1.8093,E1 25.0782,E2 510.502} C_DIS
LIN {X 45.5047,Y -86.7108,Z 95,A -67.0962,B 24.9392,C -1.8004,E1 25.0733,E2 512.509} C_DIS
LIN {X 42.3506,Y -88.2941,Z 95,A -69.059,B 24.9392,C -1.8009,E1 25.0684,E2 514.4653} C_DIS
LIN {X 39.8683,Y -89.4433,Z 95,A -70.5918,B 24.9392,C -1.8009,E1 25.0645,E2 515.9942} C_DIS
LIN {X 37.6613,Y -90.3948,Z 95,A -72.0039,B 24.9394,C -1.7987,E1 25.0608,E2 517.4084} C_DIS
LIN {X 35.4315,Y -91.2918,Z 95,A -73.4113,B 24.9394,C -1.7967,E1 25.0572,E2 518.8173} C_DIS
LIN {X 32.9908,Y -92.203,Z 95,A -74.9156,B 24.9396,C -1.7954,E1 25.0532,E2 520.3216} C_DIS
LIN {X 30.9094,Y -92.9204,Z 95,A -76.2002,B 24.9396,C -1.7939,E1 25.0498,E2 521.6071} C_DIS
LIN {X 28.6197,Y -93.6509,Z 95,A -77.6055,B 24.9398,C -1.7923,E1 25.0461,E2 523.0137} C_DIS
LIN {X 26.1185,Y -94.3801,Z 95,A -79.1234,B 24.9398,C -1.7908,E1 25.042,E2 524.5325} C_DIS
LIN {X 22.8231,Y -95.2297,Z 95,A -81.1261,B 24.9401,C -1.7884,E1 25.0366,E2 526.538} C_DIS
LIN {X 20.4791,Y -95.7611,Z 95,A -82.5295,B 24.9401,C -1.7872,E1 25.0327,E2 527.9423} C_DIS
LIN {X 18.1284,Y -96.2338,Z 95,A -83.9308,B 24.9402,C -1.7861,E1 25.0289,E2 529.3446} C_DIS
LIN {X 15.5566,Y -96.6839,Z 95,A -85.4388,B 24.9402,C -1.7857,E1 25.0248,E2 530.8522} C_DIS
LIN {X 13.1791,Y -97.0366,Z 95,A -86.8432,B 24.9402,C -1.7848,E1 25.0209,E2 532.2575} C_DIS
LIN {X 10.7938,Y -97.3308,Z 95,A -88.2477,B 24.9403,C -1.784,E1 25.017,E2 533.6627} C_DIS
LIN {X 8.4019,Y -97.5663,Z 95,A -89.6523,B 24.9403,C -1.7833,E1 25.0131,E2 535.0681} C_DIS
LIN {X 6.005,Y -97.7431,Z 95,A -91.0572,B 24.9404,C -1.7827,E1 25.0091,E2 536.4738} C_DIS
LIN {X 3.0561,Y -97.8779,Z 95,A -92.8793,B 24.9407,C -1.7787,E1 25.004,E2 538.3051} C_DIS
LIN {X 0.6684,Y -97.9224,Z 95,A -93.7835,B 24.9395,C -1.7963,E1 25.0016,E2 539.1673} C_DIS
Enddeposition()
LIN {X 0.6684,Y -97.9224,Z 95,A -93.7835,B 24.9395,C -1.7963,E1 25.0016,E2 539.1673} C_DIS
Startdeposition()
$VEL.CP = VEL_PRINT
LIN {X 2.747,Y -96.9631,Z 95,A -92.1806,B 24.9375,C -1.8264,E1 25.0063,E2 537.4933} C_DIS
LIN {X 5.7403,Y -96.8325,Z 95,A -90.4686,B 24.9375,C -1.825,E1 25.0111,E2 535.7853} C_DIS
LIN {X 9.4168,Y -96.5448,Z 95,A -88.3909,B 24.9378,C -1.8224,E1 25.0168,E2 533.7149} C_DIS
LIN {X 11.5298,Y -96.3144,Z 95,A -87.1213,B 24.9377,C -1.8236,E1 25.0204,E2 532.4432} C_DIS
LIN {X 14.6474,Y -95.8896,Z 95,A -85.1074,B 24.9372,C -1.8307,E1 25.026,E2 530.4144} C_DIS
LIN {X 17.7465,Y -95.3663,Z 95,A -83.1784,B 24.9369,C -1.8348,E1 25.0313,E2 528.4778} C_DIS
LIN {X 22.537,Y -94.3485,Z 95,A -80.6114,B 24.9375,C -1.8254,E1 25.0382,E2 525.9366} C_DIS
LIN {X 25.8725,Y -93.4895,Z 95,A -78.2939,B 24.9367,C -1.8381,E1 25.0445,E2 523.5926} C_DIS
LIN {X 29.2599,Y -92.4851,Z 95,A -76.0555,B 24.9361,C -1.8462,E1 25.0506,E2 521.339} C_DIS
LIN {X 33.2755,Y -91.1157,Z 95,A -73.7702,B 24.9365,C -1.8411,E1 25.0565,E2 519.0703} C_DIS
LIN {X 36.1666,Y -90.0083,Z 95,A -71.9015,B 24.9362,C -1.8452,E1 25.0614,E2 517.1962} C_DIS
LIN {X 40.9608,Y -87.9292,Z 95,A -68.5255,B 24.9351,C -1.8609,E1 25.0701,E2 513.7914} C_DIS
LIN {X 44.9647,Y -85.951,Z 95,A -65.6399,B 24.9341,C -1.8748,E1 25.0773,E2 510.8808} C_DIS
LIN {X 48.4675,Y -84.0253,Z 95,A -63.8377,B 24.9353,C -1.8576,E1 25.0815,E2 509.1247} C_DIS
LIN {X 51.5963,Y -82.1414,Z 95,A -61.7006,B 24.9351,C -1.8609,E1 25.0866,E2 506.9866} C_DIS
LIN {X 54.3876,Y -80.3201,Z 95,A -59.0234,B 24.9329,C -1.8922,E1 25.093,E2 504.2445} C_DIS
LIN {X 58.1273,Y -77.6568,Z 95,A -57.115,B 24.9347,C -1.8667,E1 25.0971,E2 502.4031} C_DIS
LIN {X 60.9426,Y -75.4676,Z 95,A -54.9856,B 24.9343,C -1.8722,E1 25.1018,E2 500.2686} C_DIS
LIN {X 63.2962,Y -73.5063,Z 95,A -52.24,B 24.9314,C -1.9127,E1 25.1078,E2 497.438} C_DIS
LIN {X 67.1677,Y -69.9849,Z 95,A -49.8589,B 24.9329,C -1.8923,E1 25.1125,E2 495.1151} C_DIS
LIN {X 69.7623,Y -67.3986,Z 95,A -47.9592,B 24.9332,C -1.8873,E1 25.1161,E2 493.2352} C_DIS
LIN {X 74.1687,Y -62.5172,Z 95,A -44.341,B 24.9332,C -1.8869,E1 25.1228,E2 489.6342} C_DIS
LIN {X 75.948,Y -60.3431,Z 95,A -42.4789,B 24.9324,C -1.8991,E1 25.1261,E2 487.7518} C_DIS
LIN {X 78.1156,Y -57.5096,Z 95,A -40.3975,B 24.9321,C -1.9038,E1 25.1296,E2 485.6693} C_DIS
LIN {X 80.0463,Y -54.7918,Z 95,A -38.4056,B 24.9316,C -1.9101,E1 25.1328,E2 483.6723} C_DIS
LIN {X 84.0531,Y -48.4191,Z 95,A -33.5519,B 24.9295,C -1.9389,E1 25.1399,E2 478.7755} C_DIS
LIN {X 85.6793,Y -45.4806,Z 95,A -32.0591,B 24.9305,C -1.9253,E1 25.1418,E2 477.3225} C_DIS
LIN {X 86.9118,Y -43.0774,Z 95,A -30.4196,B 24.93,C -1.9318,E1 25.1439,E2 475.6764} C_DIS
LIN {X 88.1698,Y -40.4439,Z 95,A -28.6392,B 24.9295,C -1.9392,E1 25.146,E2 473.8882} C_DIS
LIN {X 90.1246,Y -35.8759,Z 95,A -25.7647,B 24.929,C -1.9458,E1 25.1491,E2 471.0139} C_DIS
LIN {X 91.4052,Y -32.474,Z 95,A -23.6914,B 24.9287,C -1.9495,E1 25.1511,E2 468.9434} C_DIS
LIN {X 92.4576,Y -29.3466,Z 95,A -21.4946,B 24.9276,C -1.9654,E1 25.153,E2 466.7216} C_DIS
LIN {X 93.4033,Y -26.1769,Z 95,A -19.757,B 24.9278,C -1.963,E1 25.1543,E2 464.9996} C_DIS
LIN {X 94.1732,Y -23.2555,Z 95,A -18.1729,B 24.9279,C -1.9608,E1 25.1554,E2 463.4299} C_DIS
LIN {X 94.8122,Y -20.4941,Z 95,A -16.5055,B 24.9275,C -1.9659,E1 25.1564,E2 461.7603} C_DIS
LIN {X 95.2799,Y -18.196,Z 95,A -14.9637,B 24.9268,C -1.9765,E1 25.1572,E2 460.2024} C_DIS
LIN {X 95.8099,Y -15.1632,Z 95,A -13.1429,B 24.9263,C -1.9824,E1 25.1581,E2 458.3783} C_DIS
LIN {X 96.3289,Y -11.4059,Z 95,A -10.9523,B 24.9259,C -1.9876,E1 25.1588,E2 456.1883} C_DIS
LIN {X 96.6433,Y -8.3501,Z 95,A -9.296,B 24.9259,C -1.9872,E1 25.1593,E2 454.5428} C_DIS
LIN {X 96.8473,Y -5.4729,Z 95,A -7.6001,B 24.9256,C -1.9924,E1 25.1596,E2 452.8447} C_DIS
LIN {X 96.9602,Y -2.8396,Z 95,A -5.9241,B 24.9248,C -2.0021,E1 25.1598,E2 451.1558} C_DIS
LIN {X 96.9969,Y 1.0976,Z 95,A -3.7438,B 24.9248,C -2.0039,E1 25.1598,E2 448.9844} C_DIS
LIN {X 96.9422,Y 3.4278,Z 95,A -2.3894,B 24.9244,C -2.0074,E1 25.1596,E2 447.6296} C_DIS
LIN {X 96.7887,Y 6.4261,Z 95,A -0.3983,B 24.9234,C -2.0217,E1 25.1593,E2 445.6167} C_DIS
LIN {X 96.4679,Y 10.1623,Z 95,A 1.6801,B 24.9232,C -2.0233,E1 25.1588,E2 443.5466} C_DIS
LIN {X 96.0923,Y 13.2574,Z 95,A 3.5834,B 24.9226,C -2.0316,E1 25.1581,E2 441.6352} C_DIS
LIN {X 95.6133,Y 16.3574,Z 95,A 5.473,B 24.9221,C -2.0388,E1 25.1572,E2 439.7395} C_DIS
LIN {X 94.9592,Y 19.8032,Z 95,A 7.4083,B 24.922,C -2.0399,E1 25.1562,E2 437.813} C_DIS
LIN {X 94.3778,Y 22.414,Z 95,A 9.067,B 24.9214,C -2.0479,E1 25.1551,E2 436.1451} C_DIS
LIN {X 93.5882,Y 25.5074,Z 95,A 10.7869,B 24.9214,C -2.0472,E1 25.1539,E2 434.4368} C_DIS
LIN {X 92.5431,Y 29.0731,Z 95,A 13.3933,B 24.9197,C -2.0699,E1 25.1517,E2 431.7916} C_DIS
LIN {X 90.583,Y 34.7014,Z 95,A 16.3107,B 24.9207,C -2.0567,E1 25.149,E2 428.9216} C_DIS
LIN {X 89.3525,Y 37.7554,Z 95,A 18.5673,B 24.9193,C -2.0745,E1 25.1466,E2 426.6355} C_DIS
LIN {X 87.7373,Y 41.373,Z 95,A 20.7027,B 24.9194,C -2.0731,E1 25.1441,E2 424.5149} C_DIS
LIN {X 86.2649,Y 44.3593,Z 95,A 23.2086,B 24.9173,C -2.0996,E1 25.1409,E2 421.9599} C_DIS
LIN {X 84.7241,Y 47.2352,Z 95,A 25.1554,B 24.9169,C -2.1056,E1 25.1382,E2 420.009} C_DIS
LIN {X 83.0126,Y 50.1825,Z 95,A 26.9683,B 24.917,C -2.1031,E1 25.1356,E2 418.2113} C_DIS
LIN {X 81.1227,Y 53.1836,Z 95,A 28.8211,B 24.9174,C -2.0992,E1 25.1329,E2 416.377} C_DIS
LIN {X 79.3698,Y 55.7673,Z 95,A 30.6054,B 24.9172,C -2.1015,E1 25.13,E2 414.596} C_DIS
LIN {X 77.3002,Y 58.602,Z 95,A 32.5823,B 24.9171,C -2.1029,E1 25.1268,E2 412.6253} C_DIS
LIN {X 75.395,Y 61.0321,Z 95,A 34.4921,B 24.9165,C -2.1106,E1 25.1234,E2 410.7064} C_DIS
LIN {X 73.4888,Y 63.3168,Z 95,A 36.4913,B 24.9154,C -2.1239,E1 25.1198,E2 408.6848} C_DIS
LIN {X 70.3664,Y 66.7689,Z 95,A 39.0459,B 24.9155,C -2.1225,E1 25.1149,E2 406.1446} C_DIS
LIN {X 68.057,Y 69.1202,Z 95,A 40.913,B 24.9155,C -2.1236,E1 25.1112,E2 404.2827} C_DIS
LIN {X 65.8629,Y 71.2148,Z 95,A 42.9199,B 24.9145,C -2.1355,E1 25.1071,E2 402.256} C_DIS
LIN {X 63.3267,Y 73.4804,Z 95,A 44.6655,B 24.915,C -2.1294,E1 25.1035,E2 400.5317} C_DIS
LIN {X 60.9579,Y 75.4552,Z 95,A 46.535,B 24.9145,C -2.1347,E1 25.0994,E2 398.6568} C_DIS
LIN {X 58.343,Y 77.4948,Z 95,A 48.513,B 24.9142,C -2.1389,E1 25.095,E2 396.6761} C_DIS
LIN {X 55.7654,Y 79.3712,Z 95,A 50.7768,B 24.9128,C -2.1564,E1 25.0898,E2 394.3787} C_DIS
LIN {X 53.0433,Y 81.2153,Z 95,A 52.7059,B 24.9126,C -2.159,E1 25.0853,E2 392.4498} C_DIS
LIN {X 50.3099,Y 82.9352,Z 95,A 54.0652,B 24.914,C -2.1414,E1 25.0822,E2 391.1365} C_DIS
LIN {X 47.4562,Y 84.6007,Z 95,A 56.1533,B 24.9134,C -2.1492,E1 25.0771,E2 389.0361} C_DIS
LIN {X 44.886,Y 85.9925,Z 95,A 57.6969,B 24.9137,C -2.1447,E1 25.0733,E2 387.5075} C_DIS
LIN {X 42.1462,Y 87.3673,Z 95,A 59.6451,B 24.9131,C -2.1521,E1 25.0684,E2 385.5471} C_DIS
LIN {X 38.8454,Y 88.8841,Z 95,A 61.7976,B 24.9129,C -2.1547,E1 25.0629,E2 383.3936} C_DIS
LIN {X 35.2212,Y 90.3818,Z 95,A 63.9717,B 24.9131,C -2.1519,E1 25.0573,E2 381.2312} C_DIS
LIN {X 30.9932,Y 91.9171,Z 95,A 66.3731,B 24.9137,C -2.1449,E1 25.0511,E2 378.8512} C_DIS
LIN {X 28.3309,Y 92.7732,Z 95,A 68.2769,B 24.9129,C -2.1553,E1 25.0459,E2 376.9262} C_DIS
LIN {X 25.703,Y 93.5354,Z 95,A 70.0679,B 24.9123,C -2.1628,E1 25.0411,E2 375.1205} C_DIS
LIN {X 21.9535,Y 94.4849,Z 95,A 72.3476,B 24.9122,C -2.1639,E1 25.0349,E2 372.8414} C_DIS
LIN {X 18.2656,Y 95.2665,Z 95,A 74.3357,B 24.9128,C -2.1563,E1 25.0295,E2 370.8738} C_DIS
LIN {X 16.113,Y 95.6541,Z 95,A 75.8131,B 24.9122,C -2.1635,E1 25.0254,E2 369.3811} C_DIS
LIN {X 13.3094,Y 96.0849,Z 95,A 77.3486,B 24.9126,C -2.1589,E1 25.0212,E2 367.8579} C_DIS
LIN {X 10.3136,Y 96.4521,Z 95,A 79.2599,B 24.9122,C -2.1638,E1 25.0159,E2 365.9362} C_DIS
LIN {X 7.4686,Y 96.7141,Z 95,A 80.8188,B 24.9125,C -2.1593,E1 25.0115,E2 364.3888} C_DIS
LIN {X 4.457,Y 96.8997,Z 95,A 82.7722,B 24.9121,C -2.1654,E1 25.0061,E2 362.4217} C_DIS
LIN {X 1.4584,Y 96.9913,Z 95,A 84.61,B 24.9119,C -2.1675,E1 25.0009,E2 360.5793} C_DIS
LIN {X -1.5264,Y 96.99,Z 95,A 86.2933,B 24.9121,C -2.1642,E1 24.9962,E2 358.9036} C_DIS
LIN {X -5.2117,Y 96.8617,Z 95,A 88.3729,B 24.9125,C -2.16,E1 24.9905,E2 356.8335} C_DIS
LIN {X -8.1938,Y 96.6561,Z 95,A 90.1051,B 24.9126,C -2.1581,E1 24.9857,E2 355.1053} C_DIS
LIN {X -11.4244,Y 96.3267,Z 95,A 92.039,B 24.9126,C -2.1576,E1 24.9803,E2 353.1713} C_DIS
LIN {X -14.7792,Y 95.8692,Z 95,A 94.1543,B 24.9125,C -2.1603,E1 24.9744,E2 351.0478} C_DIS
LIN {X -18.2712,Y 95.2654,Z 95,A 96.2302,B 24.9126,C -2.1581,E1 24.9687,E2 348.975} C_DIS
LIN {X -21.0681,Y 94.687,Z 95,A 98.0551,B 24.9124,C -2.1614,E1 24.9637,E2 347.14} C_DIS
LIN {X -25.3978,Y 93.6178,Z 95,A 100.7628,B 24.9124,C -2.1614,E1 24.9564,E2 344.4284} C_DIS
LIN {X -29.7113,Y 92.3396,Z 95,A 102.8626,B 24.9142,C -2.1392,E1 24.9509,E2 342.3778} C_DIS
LIN {X -32.0035,Y 91.5703,Z 95,A 104.7077,B 24.9132,C -2.1517,E1 24.9459,E2 340.4994} C_DIS
LIN {X -34.7677,Y 90.5579,Z 95,A 106.2726,B 24.9138,C -2.1435,E1 24.9419,E2 338.9508} C_DIS
LIN {X -37.5867,Y 89.4236,Z 95,A 108.2223,B 24.9136,C -2.1463,E1 24.9368,E2 336.9901} C_DIS
LIN {X -41.047,Y 87.8891,Z 95,A 110.5015,B 24.9138,C -2.1444,E1 24.931,E2 334.7099} C_DIS
LIN {X -44.1318,Y 86.3812,Z 95,A 112.5752,B 24.9138,C -2.1426,E1 24.9259,E2 332.6347} C_DIS
LIN {X -46.9279,Y 84.8957,Z 95,A 114.2454,B 24.9147,C -2.1327,E1 24.9218,E2 330.9835} C_DIS
LIN {X -51.4454,Y 82.2357,Z 95,A 118.3793,B 24.9123,C -2.1623,E1 24.9118,E2 326.7663} C_DIS
LIN {X -55.6151,Y 79.4757,Z 95,A 121.1622,B 24.9133,C -2.1505,E1 24.9054,E2 324.0019} C_DIS
LIN {X -59.0782,Y 76.9359,Z 95,A 123.0092,B 24.9156,C -2.1219,E1 24.9015,E2 322.2163} C_DIS
LIN {X -61.7287,Y 74.8266,Z 95,A 124.9408,B 24.9161,C -2.1153,E1 24.8973,E2 320.2934} C_DIS
LIN {X -64.1809,Y 72.735,Z 95,A 126.9428,B 24.9161,C -2.1142,E1 24.893,E2 318.286} C_DIS
LIN {X -67.5136,Y 69.6514,Z 95,A 129.8562,B 24.9161,C -2.1156,E1 24.8871,E2 315.3572} C_DIS
LIN {X -70.7711,Y 66.3386,Z 95,A 132.3248,B 24.9173,C -2.0998,E1 24.8824,E2 312.9158} C_DIS
LIN {X -73.0718,Y 63.7953,Z 95,A 134.8552,B 24.9164,C -2.1114,E1 24.8776,E2 310.3463} C_DIS
LIN {X -75.2184,Y 61.2501,Z 95,A 136.6686,B 24.9172,C -2.1011,E1 24.8745,E2 308.549} C_DIS
LIN {X -78.6774,Y 56.7401,Z 95,A 139.5723,B 24.9191,C -2.0772,E1 24.8697,E2 305.6885} C_DIS
LIN {X -80.383,Y 54.2948,Z 95,A 141.3024,B 24.9195,C -2.0713,E1 24.8669,E2 303.9638} C_DIS
LIN {X -81.6133,Y 52.4271,Z 95,A 142.8411,B 24.9193,C -2.0747,E1 24.8646,E2 302.4092} C_DIS
LIN {X -83.1965,Y 49.8801,Z 95,A 144.7486,B 24.9193,C -2.0741,E1 24.8618,E2 300.4933} C_DIS
LIN {X -85.3354,Y 46.1219,Z 95,A 147.0141,B 24.9206,C -2.0573,E1 24.8587,E2 298.256} C_DIS
LIN {X -86.5129,Y 43.8742,Z 95,A 148.598,B 24.9208,C -2.0557,E1 24.8567,E2 296.6676} C_DIS
LIN {X -87.8224,Y 41.1903,Z 95,A 150.4878,B 24.9208,C -2.0545,E1 24.8544,E2 294.7703} C_DIS
LIN {X -89.2442,Y 38.0123,Z 95,A 152.5808,B 24.9212,C -2.0495,E1 24.8521,E2 292.6778} C_DIS
LIN {X -90.5465,Y 34.7977,Z 95,A 154.7601,B 24.9214,C -2.0475,E1 24.8498,E2 290.4911} C_DIS
LIN {X -91.6616,Y 31.7434,Z 95,A 156.4417,B 24.9224,C -2.0337,E1 24.8483,E2 288.8327} C_DIS
LIN {X -93.0207,Y 27.5042,Z 95,A 159.1435,B 24.9229,C -2.0279,E1 24.8461,E2 286.1293} C_DIS
LIN {X -93.8872,Y 24.3841,Z 95,A 161.1025,B 24.9232,C -2.0233,E1 24.8446,E2 284.1697} C_DIS
LIN {X -94.5897,Y 21.4998,Z 95,A 162.9453,B 24.9234,C -2.0207,E1 24.8434,E2 282.3225} C_DIS
LIN {X -95.4607,Y 17.2219,Z 95,A 165.2826,B 24.9247,C -2.0046,E1 24.8422,E2 280.0097} C_DIS
LIN {X -95.8535,Y 14.8807,Z 95,A 166.9831,B 24.9243,C -2.0098,E1 24.8414,E2 278.2867} C_DIS
LIN {X -96.27,Y 11.9055,Z 95,A 168.7489,B 24.9247,C -2.0038,E1 24.8408,E2 276.5247} C_DIS
LIN {X -96.6164,Y 8.6416,Z 95,A 170.6433,B 24.9253,C -1.9962,E1 24.8403,E2 274.6372} C_DIS
LIN {X -96.8878,Y 4.7346,Z 95,A 172.8383,B 24.9261,C -1.9849,E1 24.8399,E2 272.456} C_DIS
LIN {X -96.9688,Y 2.5593,Z 95,A 174.3103,B 24.926,C -1.9868,E1 24.8399,E2 270.9705} C_DIS
LIN {X -96.9976,Y -0.9969,Z 95,A 176.2796,B 24.9268,C -1.9758,E1 24.8399,E2 269.0156} C_DIS
LIN {X -96.9114,Y -4.184,Z 95,A 178.3276,B 24.9268,C -1.9751,E1 24.84,E2 266.9569} C_DIS
LIN {X -96.7367,Y -7.1838,Z 95,A 179.9123,B 24.9277,C -1.9633,E1 24.8403,E2 265.3909} C_DIS
LIN {X -96.4814,Y -10.0335,Z 95,A -178.2396,B 24.9277,C -1.9631,E1 24.8408,E2 263.5322} C_DIS
LIN {X -96.1697,Y -12.6795,Z 95,A -176.6068,B 24.928,C -1.96,E1 24.8414,E2 261.8969} C_DIS
LIN {X -95.6178,Y -16.3301,Z 95,A -174.6857,B 24.9291,C -1.9447,E1 24.8422,E2 260.0009} C_DIS
LIN {X -95.2179,Y -18.5178,Z 95,A -172.2429,B 24.9267,C -1.9777,E1 24.8436,E2 257.4648} C_DIS
LIN {X -94.1684,Y -23.275,Z 95,A -170.43,B 24.9299,C -1.9338,E1 24.8447,E2 255.7461} C_DIS
LIN {X -92.8758,Y -27.9927,Z 95,A -167.4335,B 24.9303,C -1.9285,E1 24.847,E2 252.745} C_DIS
LIN {X -92.1616,Y -30.2612,Z 95,A -165.8333,B 24.9301,C -1.9307,E1 24.8483,E2 251.1303} C_DIS
LIN {X -90.9457,Y -33.7415,Z 95,A -163.5768,B 24.9304,C -1.9269,E1 24.8505,E2 248.8701} C_DIS
LIN {X -89.6677,Y -37.0034,Z 95,A -161.5432,B 24.9309,C -1.9197,E1 24.8526,E2 246.8423} C_DIS
LIN {X -88.2889,Y -40.1812,Z 95,A -159.5774,B 24.9315,C -1.9113,E1 24.8548,E2 244.8858} C_DIS
LIN {X -86.8695,Y -43.1629,Z 95,A -157.6219,B 24.9319,C -1.906,E1 24.8572,E2 242.9323} C_DIS
LIN {X -85.0582,Y -46.6328,Z 95,A -155.4292,B 24.9326,C -1.8957,E1 24.8601,E2 240.7526} C_DIS
LIN {X -83.7611,Y -48.925,Z 95,A -153.6343,B 24.9324,C -1.8995,E1 24.8626,E2 238.9392} C_DIS
LIN {X -81.7885,Y -52.1542,Z 95,A -151.55,B 24.9331,C -1.8886,E1 24.8657,E2 236.8702} C_DIS
LIN {X -80.1756,Y -54.601,Z 95,A -149.0184,B 24.9315,C -1.9112,E1 24.8697,E2 234.2724} C_DIS
LIN {X -77.7134,Y -58.0519,Z 95,A -147.1442,B 24.9335,C -1.8838,E1 24.8728,E2 232.4544} C_DIS
LIN {X -75.8439,Y -60.4748,Z 95,A -145.53,B 24.9342,C -1.8729,E1 24.8755,E2 230.8583} C_DIS
LIN {X -71.9257,Y -65.0868,Z 95,A -141.6951,B 24.9342,C -1.8735,E1 24.8825,E2 227.0048} C_DIS
LIN {X -69.5738,Y -67.5941,Z 95,A -139.4043,B 24.9339,C -1.878,E1 24.887,E2 224.6935} C_DIS
LIN {X -67.1003,Y -70.0498,Z 95,A -137.5954,B 24.9348,C -1.8652,E1 24.8906,E2 222.9075} C_DIS
LIN {X -64.4143,Y -72.5277,Z 95,A -135.0213,B 24.9341,C -1.8751,E1 24.896,E2 220.2994} C_DIS
LIN {X -61.7852,Y -74.7797,Z 95,A -133.3357,B 24.9352,C -1.8589,E1 24.8996,E2 218.6459} C_DIS
LIN {X -59.3675,Y -76.7129,Z 95,A -131.5843,B 24.9356,C -1.853,E1 24.9034,E2 216.9022} C_DIS
LIN {X -56.8527,Y -78.5965,Z 95,A -129.6382,B 24.9356,C -1.8529,E1 24.9078,E2 214.9494} C_DIS
LIN {X -53.5804,Y -80.8611,Z 95,A -127.3567,B 24.9361,C -1.8467,E1 24.9131,E2 212.675} C_DIS
LIN {X -50.1487,Y -83.0332,Z 95,A -124.9307,B 24.9363,C -1.8441,E1 24.9188,E2 210.2477} C_DIS
LIN {X -46.9,Y -84.9113,Z 95,A -122.7554,B 24.9366,C -1.8396,E1 24.9241,E2 208.0768} C_DIS
LIN {X -43.706,Y -86.5988,Z 95,A -120.5643,B 24.9366,C -1.8389,E1 24.9296,E2 205.8814} C_DIS
LIN {X -40.4378,Y -88.1727,Z 95,A -118.3314,B 24.9366,C -1.8395,E1 24.9352,E2 203.6413} C_DIS
LIN {X -36.8894,Y -89.7141,Z 95,A -115.7965,B 24.9361,C -1.846,E1 24.9418,E2 201.0852} C_DIS
LIN {X -32.435,Y -91.4189,Z 95,A -113.3496,B 24.9372,C -1.8304,E1 24.9481,E2 198.6704} C_DIS
LIN {X -28.9807,Y -92.5717,Z 95,A -111.2087,B 24.9373,C -1.8284,E1 24.9538,E2 196.5305} C_DIS
LIN {X -25.2494,Y -93.6579,Z 95,A -108.8902,B 24.9373,C -1.8277,E1 24.9601,E2 194.2099} C_DIS
LIN {X -21.7975,Y -94.5209,Z 95,A -106.8992,B 24.9377,C -1.8226,E1 24.9654,E2 192.2282} C_DIS
LIN {X -18.457,Y -95.2296,Z 95,A -104.7867,B 24.9376,C -1.8252,E1 24.9712,E2 190.1071} C_DIS
LIN {X -14.781,Y -95.8689,Z 95,A -102.7451,B 24.938,C -1.8187,E1 24.9768,E2 188.079} C_DIS
LIN {X -12.13,Y -96.2409,Z 95,A -101.1602,B 24.938,C -1.8185,E1 24.9812,E2 186.4933} C_DIS
LIN {X -9.2132,Y -96.5636,Z 95,A -99.2012,B 24.9375,C -1.8265,E1 24.9867,E2 184.5143} C_DIS
LIN {X -5.9651,Y -96.8198,Z 95,A -97.4854,B 24.938,C -1.819,E1 24.9914,E2 182.8158} C_DIS
LIN {X -3.1545,Y -96.9506,Z 95,A -95.6945,B 24.9377,C -1.8238,E1 24.9965,E2 181.013} C_DIS
LIN {X -0.441,Y -97.0008,Z 95,A -94.1894,B 24.9379,C -1.8206,E1 25.0007,E2 179.5155} C_DIS
LIN {X -0.441,Y -97.0008,Z 95,A -94.1894,B 24.9379,C -1.8206,E1 25.0007,E2 179.5155} C_DIS
Enddeposition()
LIN {X 0.6617,Y -96.0728,Z 95,A -94.0124,B 24.9379,C -1.8197,E1 25.0011,E2 179.3406} C_DIS
Startdeposition()
$VEL.CP = VEL_PRINT
LIN {X -2.7046,Y -96.04,Z 95,A -96.4164,B 24.9389,C -1.8052,E1 24.9943,E2 181.7791} C_DIS
LIN {X -5.9253,Y -95.8965,Z 95,A -98.3702,B 24.939,C -1.804,E1 24.9889,E2 183.7364} C_DIS
LIN {X -9.3397,Y -95.6239,Z 95,A -100.4043,B 24.939,C -1.8044,E1 24.9832,E2 185.7705} C_DIS
LIN {X -11.8022,Y -95.3509,Z 95,A -101.7702,B 24.9387,C -1.8086,E1 24.9795,E2 187.1275} C_DIS
LIN {X -14.9936,Y -94.9012,Z 95,A -103.6874,B 24.9387,C -1.8092,E1 24.9742,E2 189.0448} C_DIS
LIN {X -18.1453,Y -94.3488,Z 95,A -105.6295,B 24.9387,C -1.8087,E1 24.9688,E2 190.9901} C_DIS
LIN {X -20.7652,Y -93.8075,Z 95,A -107.369,B 24.939,C -1.8044,E1 24.964,E2 192.7419} C_DIS
LIN {X -24.3789,Y -92.9346,Z 95,A -110.1057,B 24.9401,C -1.7878,E1 24.9565,E2 195.522} C_DIS
LIN {X -28.1352,Y -91.8666,Z 95,A -111.7689,B 24.9384,C -1.8123,E1 24.9522,E2 197.1299} C_DIS
LIN {X -33.1972,Y -90.1608,Z 95,A -115.2742,B 24.939,C -1.804,E1 24.9429,E2 200.6617} C_DIS
LIN {X -37.4009,Y -88.4993,Z 95,A -117.4668,B 24.9376,C -1.8238,E1 24.9373,E2 202.812} C_DIS
LIN {X -40.9416,Y -86.9191,Z 95,A -119.9894,B 24.938,C -1.8192,E1 24.9309,E2 205.3518} C_DIS
LIN {X -43.4716,Y -85.6811,Z 95,A -121.7392,B 24.938,C -1.8189,E1 24.9265,E2 207.1069} C_DIS
LIN {X -46.6244,Y -84.007,Z 95,A -123.7652,B 24.9376,C -1.8252,E1 24.9215,E2 209.1236} C_DIS
LIN {X -50.3292,Y -81.8424,Z 95,A -126.272,B 24.9372,C -1.8307,E1 24.9155,E2 211.6251} C_DIS
LIN {X -53.4597,Y -79.8326,Z 95,A -128.7699,B 24.9376,C -1.8248,E1 24.9097,E2 214.1451} C_DIS
LIN {X -56.7153,Y -77.5521,Z 95,A -130.9439,B 24.9369,C -1.8353,E1 24.9047,E2 216.3016} C_DIS
LIN {X -59.1113,Y -75.7439,Z 95,A -132.9613,B 24.9372,C -1.8309,E1 24.9002,E2 218.3367} C_DIS
LIN {X -61.7738,Y -73.5877,Z 95,A -135.128,B 24.9372,C -1.8307,E1 24.8956,E2 220.5123} C_DIS
LIN {X -65.0024,Y -70.7505,Z 95,A -137.4686,B 24.9363,C -1.8431,E1 24.8907,E2 222.8327} C_DIS
LIN {X -68.5395,Y -67.3302,Z 95,A -140.4318,B 24.936,C -1.8483,E1 24.8849,E2 225.7959} C_DIS
LIN {X -70.5442,Y -65.2271,Z 95,A -142.4714,B 24.9364,C -1.8421,E1 24.8809,E2 227.8594} C_DIS
LIN {X -74.4622,Y -60.7158,Z 95,A -145.6673,B 24.935,C -1.8622,E1 24.8752,E2 231.0218} C_DIS
LIN {X -76.5376,Y -58.0789,Z 95,A -147.8153,B 24.935,C -1.8622,E1 24.8715,E2 233.1799} C_DIS
LIN {X -79.4881,Y -53.9685,Z 95,A -150.6773,B 24.9341,C -1.8749,E1 24.867,E2 236.026} C_DIS
LIN {X -81.1438,Y -51.4482,Z 95,A -152.5684,B 24.934,C -1.8765,E1 24.8641,E2 237.9228} C_DIS
LIN {X -83.0294,Y -48.3464,Z 95,A -154.7941,B 24.9337,C -1.8802,E1 24.8609,E2 240.151} C_DIS
LIN {X -84.3251,Y -46.0466,Z 95,A -157.102,B 24.9351,C -1.8611,E1 24.8578,E2 242.5168} C_DIS
LIN {X -86.3905,Y -42.0459,Z 95,A -159.0214,B 24.9328,C -1.8929,E1 24.8554,E2 244.3706} C_DIS
LIN {X -87.7358,Y -39.1597,Z 95,A -160.9745,B 24.9326,C -1.8966,E1 24.8532,E2 246.3258} C_DIS
LIN {X -90.0301,Y -33.5527,Z 95,A -164.6181,B 24.9319,C -1.906,E1 24.8494,E2 249.9671} C_DIS
LIN {X -91.1487,Y -30.3806,Z 95,A -166.5388,B 24.9313,C -1.9147,E1 24.8477,E2 251.878} C_DIS
LIN {X -91.9835,Y -27.7521,Z 95,A -168.4465,B 24.9315,C -1.9113,E1 24.8461,E2 253.8048} C_DIS
LIN {X -93.0531,Y -23.918,Z 95,A -170.4334,B 24.9301,C -1.9308,E1 24.8447,E2 255.7567} C_DIS
LIN {X -93.8765,Y -20.4487,Z 95,A -173.0591,B 24.9308,C -1.9215,E1 24.843,E2 258.42} C_DIS
LIN {X -94.5419,Y -17.1108,Z 95,A -175.3235,B 24.9308,C -1.9205,E1 24.8419,E2 260.7003} C_DIS
LIN {X -95.0987,Y -13.6826,Z 95,A -176.9311,B 24.9293,C -1.9416,E1 24.8412,E2 262.2672} C_DIS
LIN {X -95.5189,Y -10.3539,Z 95,A -179.0015,B 24.929,C -1.9457,E1 24.8406,E2 264.3402} C_DIS
LIN {X -95.8793,Y -6.1805,Z 95,A 178.2814,B 24.929,C -1.9468,E1 24.84,E2 267.071} C_DIS
LIN {X -96.0593,Y -1.8873,Z 95,A 176.0555,B 24.9276,C -1.9656,E1 24.8398,E2 269.2654} C_DIS
LIN {X -96.0742,Y 0.9282,Z 95,A 174.3921,B 24.9271,C -1.9714,E1 24.8398,E2 270.9249} C_DIS
LIN {X -95.9747,Y 4.4619,Z 95,A 171.7646,B 24.9278,C -1.9619,E1 24.8401,E2 273.5909} C_DIS
LIN {X -95.6313,Y 9.2621,Z 95,A 169.2026,B 24.9264,C -1.9808,E1 24.8407,E2 276.1233} C_DIS
LIN {X -94.8866,Y 15.0883,Z 95,A 165.8766,B 24.9252,C -1.9976,E1 24.8419,E2 279.4291} C_DIS
LIN {X -93.7533,Y 21.0137,Z 95,A 162.0201,B 24.9249,C -2.0008,E1 24.8441,E2 283.3005} C_DIS
LIN {X -93.0611,Y 23.8868,Z 95,A 159.0941,B 24.9272,C -1.9702,E1 24.8462,E2 286.3165} C_DIS
LIN {X -91.3289,Y 29.8338,Z 95,A 156.6347,B 24.9235,C -2.0202,E1 24.8482,E2 288.671} C_DIS
LIN {X -90.45,Y 32.4044,Z 95,A 154.2282,B 24.925,C -2.0005,E1 24.8505,E2 291.138} C_DIS
LIN {X -88.8746,Y 36.5011,Z 95,A 152.3692,B 24.9226,C -2.0323,E1 24.8524,E2 292.9316} C_DIS
LIN {X -87.5265,Y 39.6244,Z 95,A 150.3893,B 24.922,C -2.0399,E1 24.8546,E2 294.9041} C_DIS
LIN {X -86.1225,Y 42.5894,Z 95,A 148.4756,B 24.9214,C -2.0471,E1 24.8569,E2 296.8111} C_DIS
LIN {X -83.3136,Y 47.8518,Z 95,A 144.7505,B 24.921,C -2.0521,E1 24.8619,E2 300.5439} C_DIS
LIN {X -81.45,Y 50.9593,Z 95,A 142.5727,B 24.9206,C -2.0577,E1 24.865,E2 302.7194} C_DIS
LIN {X -79.3638,Y 54.1521,Z 95,A 140.2663,B 24.9202,C -2.063,E1 24.8686,E2 305.0247} C_DIS
LIN {X -77.6633,Y 56.5633,Z 95,A 138.2907,B 24.9203,C -2.061,E1 24.8719,E2 307.0149} C_DIS
LIN {X -75.0256,Y 60.02,Z 95,A 135.6674,B 24.9199,C -2.0668,E1 24.8764,E2 309.6366} C_DIS
LIN {X -71.3487,Y 64.3462,Z 95,A 132.6911,B 24.9182,C -2.0886,E1 24.8817,E2 312.5745} C_DIS
LIN {X -68.9818,Y 66.8763,Z 95,A 130.3269,B 24.9185,C -2.0841,E1 24.8863,E2 314.9596} C_DIS
LIN {X -65.962,Y 69.8558,Z 95,A 127.5056,B 24.9188,C -2.0808,E1 24.892,E2 317.8006} C_DIS
LIN {X -63.5868,Y 72.0273,Z 95,A 125.7796,B 24.918,C -2.0913,E1 24.8956,E2 319.5083} C_DIS
LIN {X -59.5418,Y 75.4037,Z 95,A 122.0061,B 24.919,C -2.0779,E1 24.9039,E2 323.328} C_DIS
LIN {X -55.8729,Y 78.1612,Z 95,A 120.0755,B 24.9165,C -2.1095,E1 24.9081,E2 325.1901} C_DIS
LIN {X -52.8122,Y 80.261,Z 95,A 117.3658,B 24.9175,C -2.0977,E1 24.9145,E2 327.9368} C_DIS
LIN {X -49.9494,Y 82.0732,Z 95,A 115.5586,B 24.9166,C -2.1084,E1 24.9188,E2 329.7243} C_DIS
LIN {X -45.9879,Y 84.357,Z 95,A 112.4549,B 24.9172,C -2.1008,E1 24.9264,E2 332.855} C_DIS
LIN {X -42.5186,Y 86.1576,Z 95,A 110.6582,B 24.9155,C -2.122,E1 24.9308,E2 334.6059} C_DIS
LIN {X -38.9662,Y 87.8231,Z 95,A 108.4411,B 24.9149,C -2.1296,E1 24.9364,E2 336.8104} C_DIS
LIN {X -35.7341,Y 89.1869,Z 95,A 106.14,B 24.9153,C -2.1256,E1 24.9424,E2 339.1262} C_DIS
LIN {X -33.1694,Y 90.171,Z 95,A 104.3555,B 24.9155,C -2.1229,E1 24.9471,E2 340.9208} C_DIS
LIN {X -29.4219,Y 91.4622,Z 95,A 101.5357,B 24.9165,C -2.1106,E1 24.9547,E2 343.775} C_DIS
LIN {X -25.2489,Y 92.701,Z 95,A 100.0254,B 24.9133,C -2.1496,E1 24.9585,E2 345.195} C_DIS
LIN {X -20.6801,Y 93.826,Z 95,A 96.8301,B 24.9142,C -2.139,E1 24.9672,E2 348.4197} C_DIS
LIN {X -16.9725,Y 94.5668,Z 95,A 94.9778,B 24.9129,C -2.1545,E1 24.9722,E2 350.2373} C_DIS
LIN {X -13.0341,Y 95.1908,Z 95,A 92.369,B 24.9134,C -2.1482,E1 24.9794,E2 352.8634} C_DIS
LIN {X -9.3519,Y 95.6229,Z 95,A 89.8853,B 24.9141,C -2.1401,E1 24.9864,E2 355.3679} C_DIS
LIN {X -5.8217,Y 95.9027,Z 95,A 87.9327,B 24.9136,C -2.1464,E1 24.9918,E2 357.3062} C_DIS
LIN {X -2.3391,Y 96.051,Z 95,A 85.6326,B 24.9142,C -2.1394,E1 24.9983,E2 359.6232} C_DIS
LIN {X 1.8492,Y 96.06,Z 95,A 83.3965,B 24.9134,C -2.1489,E1 25.0044,E2 361.8366} C_DIS
LIN {X 4.9106,Y 95.953,Z 95,A 81.4762,B 24.9136,C -2.1458,E1 25.0098,E2 363.7639} C_DIS
LIN {X 8.1829,Y 95.7301,Z 95,A 79.4967,B 24.9137,C -2.1448,E1 25.0153,E2 365.7445} C_DIS
LIN {X 11.9953,Y 95.3267,Z 95,A 77.3508,B 24.9134,C -2.1494,E1 25.0212,E2 367.8782} C_DIS
LIN {X 14.69,Y 94.9481,Z 95,A 75.6532,B 24.9136,C -2.1463,E1 25.0259,E2 369.5814} C_DIS
LIN {X 17.2208,Y 94.5221,Z 95,A 73.8665,B 24.9144,C -2.1368,E1 25.0309,E2 371.3889} C_DIS
LIN {X 21.0816,Y 93.7381,Z 95,A 70.9843,B 24.916,C -2.1169,E1 25.0389,E2 374.3142} C_DIS
LIN {X 25.3491,Y 92.6739,Z 95,A 69.4233,B 24.9131,C -2.1527,E1 25.0429,E2 375.788} C_DIS
LIN {X 30.3701,Y 91.1522,Z 95,A 65.6961,B 24.915,C -2.129,E1 25.0529,E2 379.5646} C_DIS
LIN {X 34.6772,Y 89.6029,Z 95,A 62.8515,B 24.9155,C -2.1223,E1 25.0604,E2 382.419} C_DIS
LIN {X 37.6435,Y 88.3971,Z 95,A 61.4012,B 24.9144,C -2.1367,E1 25.064,E2 383.8318} C_DIS
LIN {X 40.9079,Y 86.9347,Z 95,A 59.3362,B 24.9144,C -2.1367,E1 25.0693,E2 385.8917} C_DIS
LIN {X 43.4097,Y 85.7127,Z 95,A 57.513,B 24.915,C -2.1287,E1 25.0739,E2 387.7288} C_DIS
LIN {X 47.4737,Y 83.5309,Z 95,A 54.8255,B 24.9151,C -2.1272,E1 25.0804,E2 390.412} C_DIS
LIN {X 50.6327,Y 81.6535,Z 95,A 51.6464,B 24.9182,C -2.0883,E1 25.0882,E2 393.673} C_DIS
LIN {X 55.1433,Y 78.6785,Z 95,A 49.44,B 24.9157,C -2.1197,E1 25.0931,E2 395.7977} C_DIS
LIN {X 58.6152,Y 76.1263,Z 95,A 47.3321,B 24.9147,C -2.1322,E1 25.0977,E2 397.8685} C_DIS
LIN {X 61.5792,Y 73.7496,Z 95,A 44.5728,B 24.9165,C -2.1097,E1 25.1038,E2 400.6706} C_DIS
LIN {X 66.0812,Y 69.7449,Z 95,A 41.0006,B 24.917,C -2.1033,E1 25.1112,E2 404.2435} C_DIS
LIN {X 68.5917,Y 67.2774,Z 95,A 39.1117,B 24.9168,C -2.1066,E1 25.1149,E2 406.1166} C_DIS
LIN {X 72.2371,Y 63.3466,Z 95,A 35.7908,B 24.9177,C -2.0949,E1 25.1212,E2 409.4506} C_DIS
LIN {X 75.1261,Y 59.8931,Z 95,A 33.2014,B 24.9179,C -2.0921,E1 25.1257,E2 412.0346} C_DIS
LIN {X 77.4503,Y 56.8542,Z 95,A 30.909,B 24.9184,C -2.0862,E1 25.1296,E2 414.3301} C_DIS
LIN {X 79.2286,Y 54.3519,Z 95,A 28.9159,B 24.9192,C -2.0754,E1 25.1328,E2 416.3388} C_DIS
LIN {X 81.2547,Y 51.2718,Z 95,A 26.8185,B 24.9194,C -2.0735,E1 25.136,E2 418.4301} C_DIS
LIN {X 83.1614,Y 48.1166,Z 95,A 24.0359,B 24.9215,C -2.0458,E1 25.14,E2 421.264} C_DIS
LIN {X 85.0507,Y 44.6916,Z 95,A 22.0917,B 24.9209,C -2.054,E1 25.1425,E2 423.1787} C_DIS
LIN {X 87.0458,Y 40.6692,Z 95,A 19.6567,B 24.9208,C -2.0556,E1 25.1454,E2 425.5966} C_DIS
LIN {X 88.1461,Y 38.2263,Z 95,A 18.0594,B 24.9211,C -2.0511,E1 25.1472,E2 427.196} C_DIS
LIN {X 89.662,Y 34.5246,Z 95,A 15.2526,B 24.9229,C -2.0281,E1 25.1501,E2 430.0413} C_DIS
LIN {X 90.8075,Y 31.3871,Z 95,A 13.7597,B 24.9219,C -2.0412,E1 25.1515,E2 431.4951} C_DIS
LIN {X 92.3702,Y 26.4341,Z 95,A 10.6914,B 24.9225,C -2.0329,E1 25.154,E2 434.5654} C_DIS
LIN {X 93.1896,Y 23.3866,Z 95,A 8.9481,B 24.9225,C -2.0325,E1 25.1552,E2 436.2997} C_DIS
LIN {X 94.0589,Y 19.5944,Z 95,A 6.3818,B 24.9238,C -2.0159,E1 25.1568,E2 438.8902} C_DIS
LIN {X 94.7408,Y 15.973,Z 95,A 4.3872,B 24.9238,C -2.0168,E1 25.1577,E2 440.871} C_DIS
LIN {X 95.2119,Y 12.8812,Z 95,A 2.3524,B 24.9247,C -2.0044,E1 25.1586,E2 442.9231} C_DIS
LIN {X 95.6499,Y 9.0605,Z 95,A 0.165,B 24.9249,C -2.0012,E1 25.1592,E2 445.1051} C_DIS
LIN {X 95.9216,Y 5.4784,Z 95,A -1.9069,B 24.9252,C -1.9971,E1 25.1596,E2 447.1745} C_DIS
LIN {X 96.0559,Y 2.0727,Z 95,A -3.9471,B 24.9257,C -1.9902,E1 25.1598,E2 449.2186} C_DIS
LIN {X 96.0754,Y -0.6852,Z 95,A -5.871,B 24.9269,C -1.9742,E1 25.1598,E2 451.1687} C_DIS
LIN {X 95.9505,Y -4.9568,Z 95,A -8.1561,B 24.9268,C -1.9761,E1 25.1595,E2 453.4358} C_DIS
LIN {X 95.7203,Y -8.2982,Z 95,A -10.166,B 24.9273,C -1.9692,E1 25.1591,E2 455.4501} C_DIS
LIN {X 95.3896,Y -11.4833,Z 95,A -12.1373,B 24.9279,C -1.9607,E1 25.1584,E2 457.4299} C_DIS
LIN {X 94.7633,Y -15.8383,Z 95,A -14.5354,B 24.9279,C -1.961,E1 25.1574,E2 459.8132} C_DIS
LIN {X 94.2217,Y -18.8013,Z 95,A -16.4709,B 24.9287,C -1.9498,E1 25.1564,E2 461.7636} C_DIS
LIN {X 93.5099,Y -22.0692,Z 95,A -18.3902,B 24.929,C -1.9464,E1 25.1552,E2 463.68} C_DIS
LIN {X 92.7492,Y -25.0706,Z 95,A -20.15,B 24.9292,C -1.9439,E1 25.154,E2 465.4355} C_DIS
LIN {X 90.9741,Y -30.8983,Z 95,A -24.608,B 24.9323,C -1.901,E1 25.1501,E2 469.9694} C_DIS
LIN {X 89.4251,Y -35.1296,Z 95,A -26.7677,B 24.9314,C -1.9128,E1 25.148,E2 472.0893} C_DIS
LIN {X 87.5233,Y -39.6315,Z 95,A -29.2936,B 24.931,C -1.9188,E1 25.1452,E2 474.5871} C_DIS
LIN {X 86.1342,Y -42.566,Z 95,A -31.284,B 24.9315,C -1.9109,E1 25.1428,E2 476.5855} C_DIS
LIN {X 84.9943,Y -44.7985,Z 95,A -33.0594,B 24.9326,C -1.8958,E1 25.1404,E2 478.3872} C_DIS
LIN {X 83.1666,Y -48.1076,Z 95,A -35.4623,B 24.9335,C -1.8836,E1 25.1371,E2 480.8064} C_DIS
LIN {X 80.4455,Y -52.5324,Z 95,A -38.5417,B 24.9341,C -1.8755,E1 25.1325,E2 483.8894} C_DIS
LIN {X 78.6508,Y -55.183,Z 95,A -40.0651,B 24.9334,C -1.8849,E1 25.1301,E2 485.3833} C_DIS
LIN {X 76.7038,Y -57.8576,Z 95,A -41.9199,B 24.9334,C -1.884,E1 25.127,E2 487.2313} C_DIS
LIN {X 74.0266,Y -61.2458,Z 95,A -44.6117,B 24.9343,C -1.8727,E1 25.1223,E2 489.937} C_DIS
LIN {X 70.3508,Y -65.4369,Z 95,A -47.8306,B 24.9346,C -1.8682,E1 25.1163,E2 493.1523} C_DIS
LIN {X 67.4873,Y -68.3843,Z 95,A -50.1817,B 24.9347,C -1.866,E1 25.1117,E2 495.4986} C_DIS
LIN {X 65.6019,Y -70.1954,Z 95,A -52.5098,B 24.937,C -1.8335,E1 25.1068,E2 497.8941} C_DIS
LIN {X 62.5221,Y -72.9522,Z 95,A -54.2422,B 24.9355,C -1.8552,E1 25.1033,E2 499.5682} C_DIS
LIN {X 60.2758,Y -74.8188,Z 95,A -55.7595,B 24.9352,C -1.8598,E1 25.1,E2 501.0689} C_DIS
LIN {X 58.2856,Y -76.3802,Z 95,A -57.7911,B 24.9367,C -1.837,E1 25.0954,E2 503.147} C_DIS
LIN {X 53.7792,Y -79.6163,Z 95,A -60.8345,B 24.9365,C -1.8402,E1 25.0885,E2 506.1724} C_DIS
LIN {X 50.5492,Y -81.7062,Z 95,A -63.2613,B 24.9372,C -1.8308,E1 25.0828,E2 508.6135} C_DIS
LIN {X 47.1288,Y -83.7253,Z 95,A -65.6613,B 24.9375,C -1.8254,E1 25.0769,E2 511.019} C_DIS
LIN {X 43.4341,Y -85.7002,Z 95,A -68.3573,B 24.9383,C -1.8139,E1 25.0702,E2 513.7348} C_DIS
LIN {X 38.5468,Y -88.0064,Z 95,A -71.2551,B 24.9379,C -1.8209,E1 25.0629,E2 516.6088} C_DIS
LIN {X 35.0391,Y -89.4607,Z 95,A -73.3948,B 24.9378,C -1.8223,E1 25.0574,E2 518.7403} C_DIS
LIN {X 31.4863,Y -90.7727,Z 95,A -76.5142,B 24.9401,C -1.7881,E1 25.049,E2 521.9344} C_DIS
LIN {X 26.9792,Y -92.2128,Z 95,A -79.2704,B 24.9401,C -1.7872,E1 25.0416,E2 524.6879} C_DIS
LIN {X 22.6408,Y -93.3721,Z 95,A -81.3278,B 24.9388,C -1.8069,E1 25.0362,E2 526.6956} C_DIS
LIN {X 18.2045,Y -94.3374,Z 95,A -83.8128,B 24.9384,C -1.8126,E1 25.0294,E2 529.1641} C_DIS
LIN {X 15.1271,Y -94.8806,Z 95,A -85.7377,B 24.9387,C -1.8089,E1 25.0241,E2 531.0957} C_DIS
LIN {X 11.929,Y -95.3353,Z 95,A -87.822,B 24.9391,C -1.802,E1 25.0183,E2 533.1946} C_DIS
LIN {X 9.1536,Y -95.6413,Z 95,A -89.5249,B 24.9393,C -1.7997,E1 25.0135,E2 534.9019} C_DIS
LIN {X 4.6816,Y -95.9653,Z 95,A -92.0109,B 24.9389,C -1.8053,E1 25.0066,E2 537.3738} C_DIS
LIN {X 1.3462,Y -96.0693,Z 95,A -93.9786,B 24.9389,C -1.8055,E1 25.0011,E2 539.3406} C_DIS
LIN {X 1.3462,Y -96.0693,Z 95,A -93.9786,B 24.9389,C -1.8055,E1 25.0011,E2 539.3406} C_DIS
Enddeposition()
LIN {X 0.656,Y -95.1517,Z 95,A -93.995,B 24.9368,C -1.8356,E1 25.0013,E2 539.2856} C_DIS
Startdeposition()
$VEL.CP = VEL_PRINT
LIN {X 4.5205,Y -95.0475,Z 95,A -91.1566,B 24.9355,C -1.8545,E1 25.0093,E2 536.4029} C_DIS
LIN {X 9.5304,Y -94.6762,Z 95,A -88.3962,B 24.9361,C -1.8465,E1 25.017,E2 533.6629} C_DIS
LIN {X 13.1053,Y -94.2475,Z 95,A -86.0214,B 24.9355,C -1.8553,E1 25.0236,E2 531.2691} C_DIS
LIN {X 16.2714,Y -93.7538,Z 95,A -84.0251,B 24.9352,C -1.8592,E1 25.0291,E2 529.2657} C_DIS
Enddeposition()
END
